RoboDK station: 07252019 KR10 2 Script Print.rdk

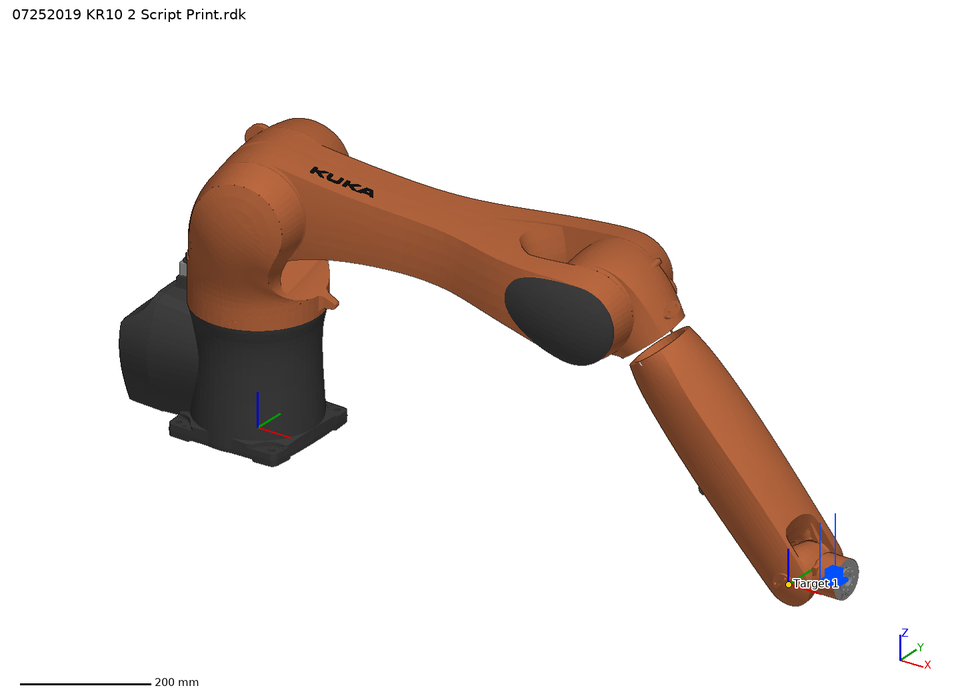
[picture v0: the station drawn from its stored meshes, robots at their saved joint values, targets as dots, program paths as lines]
Station 07252019 KR10 2 Script Print. Poses are relative to the parent item; angles as X-Y-Z fixed-axis rotations.
  - frame KUKA KR 10 R1100 sixx Base at (0, 0, 0) mm
    - robot KUKA KR 10 R1100 sixx: 6 axes, payload 10 kg, reach 1101 mm, repeatability 0.03 mm, weight 54 kg
        modified DH rows (alpha deg, a mm, theta deg, d mm): 0, 0, 0, 400; -90, 25, 0, 0; 0, 560, -90, 0; -90, 35, 0, 515; 90, 0, 0, 0; -90, 0, 180, 80
        joint limits [-170, -190, -120, -185, -120, -350] to [170, 45, 156, 185, 120, 350]; home [0, -90, 90, 0, 0, 0]; saved at [-10.597, 6.174, 47.039, 166.851, 53.94, -172.17]
    - target Target 1 (Cartesian target) at (915.91, 105.12, -52.31) mm, rotated rx -159.1 ry 89.96 rz -159.1 deg; joints [-7.168, 0.501, 63.462, 172.028, 64.143, -176.495] of KUKA KR 10 R1100 sixx
  - frame Frame 2 at (915.91, 105.12, -52.31) mm
  - machining project Print3D settings: C:/Users/Rez/Downloads/XYZ_20mm_Calibration_Cube/files/CFFFP_xyzCalibration_cube.gcode | rotZ(0) | rotX(0)*rotY(0)
  - Python program Extruder (listed below)
  - Python program M_RunCode (listed below)
  - program Print3D (7039 instructions, listed below)
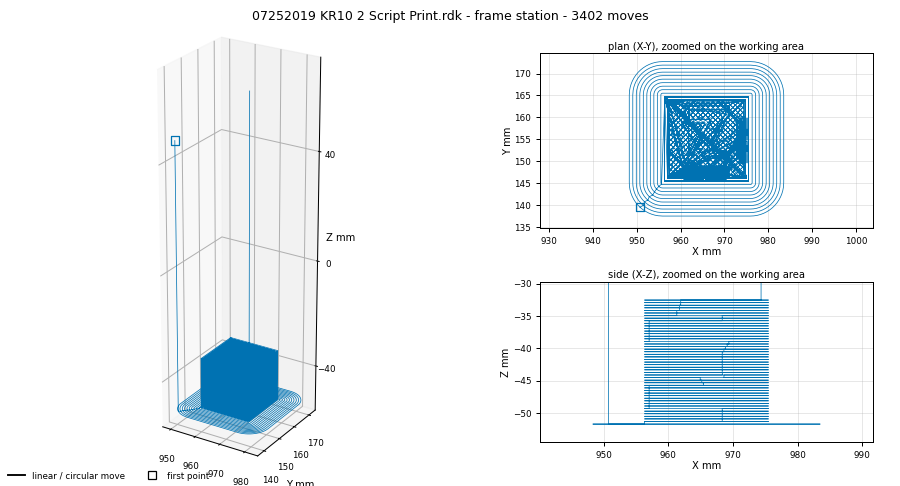
[picture p0: tool path of 07252019 KR10 2 Script Print.rdk in frame station, 3402 of 3402 moves have a stored position in this frame; points joined in program order, loops and branches not executed]

--- Python program Extruder ---
# -*- coding: utf-8 -*-
"""
Created on Fri May 24 11:08:35 2019

@author: Rez
"""

import telnetlib
import sys

tn = telnetlib.Telnet('192.168.1.112', 23)
tn.read_until(b"Smoothie command shell")
str1 = str(sys.argv[1])
str2 = "G1 E" + str1 + "\n"
str3 = str2.encode('utf-8')
tn.write(str3)
tn.read_until(b"ok")
tn.write(b"exit")
tn.close
exit

--- Python program M_RunCode ---
# -*- coding: utf-8 -*-
"""
Created on Fri May 24 11:08:35 2019

@author: Rez
"""

import telnetlib
import sys

tn = telnetlib.Telnet('192.168.1.112', 23)
tn.read_until(b"Smoothie command shell")
str1 = str(sys.argv[1])
str4 = str(sys.argv[2])
str2 = "M" + str1 + " P" +str4 + "\n"
str3 = str2.encode('utf-8')
tn.write(str3)
tn.read_until(b"ok")
tn.write(b"exit")
tn.close
exit

--- program Print3D (robot KUKA KR 10 R1100 sixx) ---
  Accurate (rounding -1 mm)
  Set Ref.: Frame 2
  Set Tool at (0, 0, 0) mm
  Call M_RunCode(104,0)
  Call M_RunCode(105,0)
  Call M_RunCode(109,0)
  Call M_RunCode(82,0)
  Call Extruder(0.000)
  Set speed (3.3 mm/s)
  Call Extruder(0.000)
  Set speed (1000.0 mm/s)
  MoveJ 1 to (34.82, 34.44, 100.6) mm, rotated rx 0 ry 90 rz 0 deg; joints [-9.106, -6.941, 65.166, 169.323, 58.671, -174.401]
  MoveL 2 to (34.82, 34.44, 100.6) mm, rotated rx 0 ry 90 rz 0 deg; joints [-9.106, -6.941, 65.166, 169.323, 58.671, -174.401]
  MoveL 3 to (34.82, 34.44, 0.6) mm, rotated rx 0 ry 90 rz 0 deg; joints [-9.106, 3.069, 55.606, 169.373, 59.113, -174.498]
  MoveL 4 to (34.82, 34.44, 0.6) mm, rotated rx 0 ry 90 rz 0 deg; joints [-9.106, 3.069, 55.606, 169.373, 59.113, -174.498]
  Call Extruder(0.000)
  Call Extruder(0.000)
  Call Extruder(0.000)
  Set speed (30.0 mm/s)
  Call Extruder(0.000)
  MoveL 5 to (34.82, 34.44, 0.6) mm, rotated rx 0 ry 90 rz 0 deg; joints [-9.106, 3.069, 55.606, 169.373, 59.113, -174.498]
  Call M_RunCode(107,0)
  Set speed (60.0 mm/s)
  MoveL 6 to (34.82, 34.44, 0.6) mm, rotated rx 0 ry 90 rz 0 deg; joints [-9.106, 3.069, 55.606, 169.373, 59.113, -174.498]
  Set speed (30.0 mm/s)
  Call Extruder(0.000)
  MoveL 7 to (34.82, 34.44, 0.6) mm, rotated rx 0 ry 90 rz 0 deg; joints [-9.106, 3.069, 55.606, 169.373, 59.113, -174.498]
  Call Extruder(0.156)
  MoveL 8 to (35.42, 33.94, 0.6) mm, rotated rx 0 ry 90 rz 0 deg; joints [-9.068, 3.107, 55.496, 169.409, 59.039, -174.506]
  Call Extruder(0.311)
  MoveL 9 to (36.06, 33.5, 0.6) mm, rotated rx 0 ry 90 rz 0 deg; joints [-9.033, 3.15, 55.372, 169.441, 58.956, -174.509]
  Call Extruder(0.467)
  MoveL 10 to (36.75, 33.13, 0.6) mm, rotated rx 0 ry 90 rz 0 deg; joints [-9.002, 3.197, 55.237, 169.467, 58.867, -174.509]
  Call Extruder(0.622)
  MoveL 11 to (37.47, 32.83, 0.6) mm, rotated rx 0 ry 90 rz 0 deg; joints [-8.976, 3.248, 55.092, 169.487, 58.772, -174.504]
  Call Extruder(0.778)
  MoveL 12 to (38.22, 32.61, 0.6) mm, rotated rx 0 ry 90 rz 0 deg; joints [-8.954, 3.302, 54.938, 169.501, 58.671, -174.496]
  Call Extruder(0.933)
  MoveL 13 to (38.98, 32.47, 0.6) mm, rotated rx 0 ry 90 rz 0 deg; joints [-8.938, 3.358, 54.777, 169.509, 58.566, -174.484]
  Call Extruder(1.137)
  MoveL 14 to (40, 32.4, 0.6) mm, rotated rx 0 ry 90 rz 0 deg; joints [-8.923, 3.435, 54.558, 169.51, 58.425, -174.463]
  Call Extruder(5.128)
  MoveL 15 to (60, 32.4, 0.6) mm, rotated rx 0 ry 90 rz 0 deg; joints [-8.727, 5.076, 49.99, 169.395, 55.528, -173.951]
  Call Extruder(5.284)
  MoveL 16 to (60.78, 32.44, 0.6) mm, rotated rx 0 ry 90 rz 0 deg; joints [-8.722, 5.145, 49.802, 169.386, 55.411, -173.927]
  Call Extruder(5.439)
  MoveL 17 to (61.55, 32.56, 0.6) mm, rotated rx 0 ry 90 rz 0 deg; joints [-8.722, 5.215, 49.612, 169.37, 55.293, -173.9]
  Call Extruder(5.595)
  MoveL 18 to (62.3, 32.76, 0.6) mm, rotated rx 0 ry 90 rz 0 deg; joints [-8.727, 5.285, 49.422, 169.349, 55.175, -173.87]
  Call Extruder(5.750)
  MoveL 19 to (63.03, 33.03, 0.6) mm, rotated rx 0 ry 90 rz 0 deg; joints [-8.737, 5.355, 49.234, 169.321, 55.06, -173.836]
  Call Extruder(5.906)
  MoveL 20 to (63.73, 33.38, 0.6) mm, rotated rx 0 ry 90 rz 0 deg; joints [-8.752, 5.423, 49.051, 169.288, 54.948, -173.8]
  Call Extruder(6.061)
  MoveL 21 to (64.39, 33.8, 0.6) mm, rotated rx 0 ry 90 rz 0 deg; joints [-8.772, 5.488, 48.874, 169.25, 54.841, -173.761]
  Call Extruder(6.217)
  MoveL 22 to (65, 34.28, 0.6) mm, rotated rx 0 ry 90 rz 0 deg; joints [-8.796, 5.551, 48.705, 169.206, 54.739, -173.719]
  Call Extruder(6.372)
  MoveL 23 to (65.56, 34.82, 0.6) mm, rotated rx 0 ry 90 rz 0 deg; joints [-8.824, 5.61, 48.546, 169.159, 54.644, -173.676]
  Call Extruder(6.528)
  MoveL 24 to (66.06, 35.42, 0.6) mm, rotated rx 0 ry 90 rz 0 deg; joints [-8.856, 5.665, 48.398, 169.107, 54.557, -173.632]
  Call Extruder(6.684)
  MoveL 25 to (66.5, 36.06, 0.6) mm, rotated rx 0 ry 90 rz 0 deg; joints [-8.892, 5.714, 48.265, 169.052, 54.478, -173.587]
  Call Extruder(6.839)
  MoveL 26 to (66.87, 36.75, 0.6) mm, rotated rx 0 ry 90 rz 0 deg; joints [-8.931, 5.759, 48.146, 168.994, 54.41, -173.542]
  Call Extruder(6.995)
  MoveL 27 to (67.17, 37.47, 0.6) mm, rotated rx 0 ry 90 rz 0 deg; joints [-8.973, 5.797, 48.044, 168.935, 54.351, -173.498]
  Call Extruder(7.150)
  MoveL 28 to (67.39, 38.22, 0.6) mm, rotated rx 0 ry 90 rz 0 deg; joints [-9.017, 5.829, 47.959, 168.873, 54.304, -173.453]
  Call Extruder(7.306)
  MoveL 29 to (67.53, 38.98, 0.6) mm, rotated rx 0 ry 90 rz 0 deg; joints [-9.063, 5.854, 47.892, 168.811, 54.268, -173.411]
  Call Extruder(7.509)
  MoveL 30 to (67.6, 40, 0.6) mm, rotated rx 0 ry 90 rz 0 deg; joints [-9.125, 5.875, 47.834, 168.73, 54.24, -173.358]
  Call Extruder(11.501)
  MoveL 31 to (67.6, 60, 0.6) mm, rotated rx 0 ry 90 rz 0 deg; joints [-10.357, 6.202, 46.965, 167.138, 53.863, -172.331]
  Call Extruder(11.656)
  MoveL 32 to (67.56, 60.78, 0.6) mm, rotated rx 0 ry 90 rz 0 deg; joints [-10.405, 6.212, 46.939, 167.076, 53.853, -172.292]
  Call Extruder(11.812)
  MoveL 33 to (67.44, 61.55, 0.6) mm, rotated rx 0 ry 90 rz 0 deg; joints [-10.454, 6.214, 46.933, 167.016, 53.856, -172.255]
  Call Extruder(11.967)
  MoveL 34 to (67.24, 62.3, 0.6) mm, rotated rx 0 ry 90 rz 0 deg; joints [-10.502, 6.208, 46.948, 166.958, 53.872, -172.223]
  Call Extruder(12.123)
  MoveL 35 to (66.97, 63.03, 0.6) mm, rotated rx 0 ry 90 rz 0 deg; joints [-10.55, 6.195, 46.983, 166.903, 53.9, -172.194]
  Call Extruder(12.278)
  MoveL 36 to (66.62, 63.73, 0.6) mm, rotated rx 0 ry 90 rz 0 deg; joints [-10.597, 6.174, 47.039, 166.851, 53.94, -172.17]
  Call Extruder(12.434)
  MoveL 37 to (66.21, 64.39, 0.6) mm, rotated rx 0 ry 90 rz 0 deg; joints [-10.642, 6.146, 47.113, 166.803, 53.991, -172.151]
  Call Extruder(12.589)
  MoveL 38 to (65.72, 65, 0.6) mm, rotated rx 0 ry 90 rz 0 deg; joints [-10.685, 6.111, 47.207, 166.76, 54.054, -172.136]
  Call Extruder(12.745)
  MoveL 39 to (65.18, 65.56, 0.6) mm, rotated rx 0 ry 90 rz 0 deg; joints [-10.726, 6.069, 47.317, 166.722, 54.126, -172.127]
  Call Extruder(12.901)
  MoveL 40 to (64.58, 66.06, 0.6) mm, rotated rx 0 ry 90 rz 0 deg; joints [-10.764, 6.022, 47.443, 166.689, 54.209, -172.122]
  Call Extruder(13.056)
  MoveL 41 to (63.94, 66.5, 0.6) mm, rotated rx 0 ry 90 rz 0 deg; joints [-10.798, 5.969, 47.585, 166.662, 54.299, -172.123]
  Call Extruder(13.212)
  MoveL 42 to (63.25, 66.87, 0.6) mm, rotated rx 0 ry 90 rz 0 deg; joints [-10.829, 5.911, 47.739, 166.64, 54.397, -172.128]
  Call Extruder(13.367)
  MoveL 43 to (62.53, 67.17, 0.6) mm, rotated rx 0 ry 90 rz 0 deg; joints [-10.856, 5.849, 47.905, 166.625, 54.502, -172.139]
  Call Extruder(13.523)
  MoveL 44 to (61.78, 67.39, 0.6) mm, rotated rx 0 ry 90 rz 0 deg; joints [-10.878, 5.783, 48.08, 166.615, 54.612, -172.154]
  Call Extruder(13.678)
  MoveL 45 to (61.02, 67.53, 0.6) mm, rotated rx 0 ry 90 rz 0 deg; joints [-10.896, 5.715, 48.263, 166.612, 54.726, -172.174]
  Call Extruder(13.882)
  MoveL 46 to (60, 67.6, 0.6) mm, rotated rx 0 ry 90 rz 0 deg; joints [-10.912, 5.623, 48.511, 166.618, 54.879, -172.207]
  Call Extruder(17.873)
  MoveL 47 to (40, 67.6, 0.6) mm, rotated rx 0 ry 90 rz 0 deg; joints [-11.155, 3.921, 53.184, 166.784, 57.802, -172.867]
  Call Extruder(18.029)
  MoveL 48 to (39.22, 67.56, 0.6) mm, rotated rx 0 ry 90 rz 0 deg; joints [-11.162, 3.859, 53.359, 166.792, 57.913, -172.893]
  Call Extruder(18.184)
  MoveL 49 to (38.45, 67.44, 0.6) mm, rotated rx 0 ry 90 rz 0 deg; joints [-11.164, 3.796, 53.535, 166.805, 58.024, -172.922]
  Call Extruder(18.340)
  MoveL 50 to (37.7, 67.24, 0.6) mm, rotated rx 0 ry 90 rz 0 deg; joints [-11.161, 3.734, 53.71, 166.825, 58.133, -172.955]
  Call Extruder(18.495)
  MoveL 51 to (36.97, 66.97, 0.6) mm, rotated rx 0 ry 90 rz 0 deg; joints [-11.153, 3.673, 53.882, 166.85, 58.24, -172.99]
  Call Extruder(18.651)
  MoveL 52 to (36.27, 66.62, 0.6) mm, rotated rx 0 ry 90 rz 0 deg; joints [-11.14, 3.614, 54.05, 166.881, 58.345, -173.027]
  Call Extruder(18.806)
  MoveL 53 to (35.61, 66.2, 0.6) mm, rotated rx 0 ry 90 rz 0 deg; joints [-11.122, 3.557, 54.212, 166.917, 58.444, -173.066]
  Call Extruder(18.962)
  MoveL 54 to (35, 65.72, 0.6) mm, rotated rx 0 ry 90 rz 0 deg; joints [-11.099, 3.502, 54.366, 166.957, 58.539, -173.106]
  Call Extruder(19.117)
  MoveL 55 to (34.44, 65.18, 0.6) mm, rotated rx 0 ry 90 rz 0 deg; joints [-11.071, 3.452, 54.51, 167.002, 58.627, -173.148]
  Call Extruder(19.273)
  MoveL 56 to (33.94, 64.58, 0.6) mm, rotated rx 0 ry 90 rz 0 deg; joints [-11.04, 3.405, 54.644, 167.051, 58.708, -173.19]
  Call Extruder(19.429)
  MoveL 57 to (33.5, 63.94, 0.6) mm, rotated rx 0 ry 90 rz 0 deg; joints [-11.004, 3.362, 54.766, 167.103, 58.781, -173.232]
  Call Extruder(19.584)
  MoveL 58 to (33.13, 63.25, 0.6) mm, rotated rx 0 ry 90 rz 0 deg; joints [-10.965, 3.324, 54.874, 167.158, 58.845, -173.273]
  Call Extruder(19.740)
  MoveL 59 to (32.83, 62.53, 0.6) mm, rotated rx 0 ry 90 rz 0 deg; joints [-10.923, 3.291, 54.968, 167.215, 58.899, -173.315]
  Call Extruder(19.895)
  MoveL 60 to (32.61, 61.78, 0.6) mm, rotated rx 0 ry 90 rz 0 deg; joints [-10.878, 3.264, 55.047, 167.274, 58.944, -173.355]
  Call Extruder(20.051)
  MoveL 61 to (32.47, 61.02, 0.6) mm, rotated rx 0 ry 90 rz 0 deg; joints [-10.831, 3.242, 55.109, 167.333, 58.978, -173.393]
  Call Extruder(20.254)
  MoveL 62 to (32.4, 60, 0.6) mm, rotated rx 0 ry 90 rz 0 deg; joints [-10.767, 3.222, 55.166, 167.412, 59.007, -173.441]
  Call Extruder(24.246)
  MoveL 63 to (32.4, 40, 0.6) mm, rotated rx 0 ry 90 rz 0 deg; joints [-9.488, 2.957, 55.927, 168.954, 59.357, -174.318]
  Call Extruder(24.401)
  MoveL 64 to (32.44, 39.22, 0.6) mm, rotated rx 0 ry 90 rz 0 deg; joints [-9.438, 2.951, 55.946, 169.013, 59.364, -174.35]
  Call Extruder(24.557)
  MoveL 65 to (32.56, 38.45, 0.6) mm, rotated rx 0 ry 90 rz 0 deg; joints [-9.387, 2.95, 55.948, 169.072, 59.36, -174.38]
  Call Extruder(24.712)
  MoveL 66 to (32.76, 37.7, 0.6) mm, rotated rx 0 ry 90 rz 0 deg; joints [-9.337, 2.956, 55.933, 169.129, 59.345, -174.408]
  Call Extruder(24.868)
  MoveL 67 to (33.03, 36.97, 0.6) mm, rotated rx 0 ry 90 rz 0 deg; joints [-9.287, 2.967, 55.9, 169.185, 59.319, -174.433]
  Call Extruder(25.023)
  MoveL 68 to (33.38, 36.27, 0.6) mm, rotated rx 0 ry 90 rz 0 deg; joints [-9.239, 2.984, 55.85, 169.237, 59.283, -174.454]
  Call Extruder(25.179)
  MoveL 69 to (33.79, 35.61, 0.6) mm, rotated rx 0 ry 90 rz 0 deg; joints [-9.192, 3.007, 55.784, 169.286, 59.236, -174.472]
  Call Extruder(25.334)
  MoveL 70 to (34.28, 35, 0.6) mm, rotated rx 0 ry 90 rz 0 deg; joints [-9.148, 3.035, 55.702, 169.332, 59.179, -174.487]
  Call Extruder(25.490)
  MoveL 71 to (34.82, 34.44, 0.6) mm, rotated rx 0 ry 90 rz 0 deg; joints [-9.106, 3.069, 55.606, 169.373, 59.113, -174.498]
  Set speed (60.0 mm/s)
  MoveL 72 to (35.6, 34.81, 0.6) mm, rotated rx 0 ry 90 rz 0 deg; joints [-9.122, 3.132, 55.425, 169.342, 58.999, -174.463]
  Set speed (30.0 mm/s)
  Call Extruder(25.637)
  MoveL 73 to (36.19, 34.37, 0.6) mm, rotated rx 0 ry 90 rz 0 deg; joints [-9.087, 3.17, 55.315, 169.374, 58.925, -174.469]
  Call Extruder(25.784)
  MoveL 74 to (36.82, 33.99, 0.6) mm, rotated rx 0 ry 90 rz 0 deg; joints [-9.057, 3.213, 55.192, 169.401, 58.843, -174.47]
  Call Extruder(25.931)
  MoveL 75 to (37.49, 33.68, 0.6) mm, rotated rx 0 ry 90 rz 0 deg; joints [-9.03, 3.26, 55.058, 169.422, 58.755, -174.467]
  Call Extruder(26.078)
  MoveL 76 to (38.19, 33.45, 0.6) mm, rotated rx 0 ry 90 rz 0 deg; joints [-9.008, 3.31, 54.915, 169.437, 58.661, -174.46]
  Call Extruder(26.226)
  MoveL 77 to (38.91, 33.29, 0.6) mm, rotated rx 0 ry 90 rz 0 deg; joints [-8.991, 3.363, 54.764, 169.446, 58.563, -174.45]
  Call Extruder(26.443)
  MoveL 78 to (40, 33.2, 0.6) mm, rotated rx 0 ry 90 rz 0 deg; joints [-8.974, 3.445, 54.53, 169.449, 58.413, -174.427]
  Call Extruder(30.435)
  MoveL 79 to (60, 33.2, 0.6) mm, rotated rx 0 ry 90 rz 0 deg; joints [-8.777, 5.087, 49.961, 169.332, 55.515, -173.912]
  Call Extruder(30.582)
  MoveL 80 to (60.74, 33.24, 0.6) mm, rotated rx 0 ry 90 rz 0 deg; joints [-8.772, 5.153, 49.782, 169.323, 55.404, -173.89]
  Call Extruder(30.729)
  MoveL 81 to (61.46, 33.36, 0.6) mm, rotated rx 0 ry 90 rz 0 deg; joints [-8.773, 5.219, 49.602, 169.308, 55.292, -173.864]
  Call Extruder(30.876)
  MoveL 82 to (62.17, 33.56, 0.6) mm, rotated rx 0 ry 90 rz 0 deg; joints [-8.778, 5.285, 49.423, 169.287, 55.182, -173.835]
  Call Extruder(31.023)
  MoveL 83 to (62.86, 33.83, 0.6) mm, rotated rx 0 ry 90 rz 0 deg; joints [-8.789, 5.35, 49.246, 169.26, 55.073, -173.802]
  Call Extruder(31.170)
  MoveL 84 to (63.51, 34.18, 0.6) mm, rotated rx 0 ry 90 rz 0 deg; joints [-8.804, 5.414, 49.074, 169.227, 54.968, -173.767]
  Call Extruder(31.317)
  MoveL 85 to (64.12, 34.59, 0.6) mm, rotated rx 0 ry 90 rz 0 deg; joints [-8.824, 5.475, 48.909, 169.189, 54.869, -173.729]
  Call Extruder(31.464)
  MoveL 86 to (64.68, 35.07, 0.6) mm, rotated rx 0 ry 90 rz 0 deg; joints [-8.848, 5.533, 48.753, 169.147, 54.775, -173.69]
  Call Extruder(31.612)
  MoveL 87 to (65.19, 35.6, 0.6) mm, rotated rx 0 ry 90 rz 0 deg; joints [-8.876, 5.587, 48.608, 169.1, 54.688, -173.649]
  Call Extruder(31.759)
  MoveL 88 to (65.63, 36.19, 0.6) mm, rotated rx 0 ry 90 rz 0 deg; joints [-8.908, 5.636, 48.475, 169.05, 54.61, -173.607]
  Call Extruder(31.906)
  MoveL 89 to (66.01, 36.82, 0.6) mm, rotated rx 0 ry 90 rz 0 deg; joints [-8.944, 5.68, 48.356, 168.996, 54.541, -173.564]
  Call Extruder(32.053)
  MoveL 90 to (66.32, 37.49, 0.6) mm, rotated rx 0 ry 90 rz 0 deg; joints [-8.982, 5.719, 48.253, 168.941, 54.482, -173.522]
  Call Extruder(32.200)
  MoveL 91 to (66.56, 38.19, 0.6) mm, rotated rx 0 ry 90 rz 0 deg; joints [-9.023, 5.751, 48.168, 168.883, 54.433, -173.48]
  Call Extruder(32.347)
  MoveL 92 to (66.71, 38.91, 0.6) mm, rotated rx 0 ry 90 rz 0 deg; joints [-9.067, 5.776, 48.1, 168.825, 54.396, -173.439]
  Call Extruder(32.565)
  MoveL 93 to (66.8, 40, 0.6) mm, rotated rx 0 ry 90 rz 0 deg; joints [-9.133, 5.801, 48.034, 168.738, 54.364, -173.382]
  Call Extruder(36.556)
  MoveL 94 to (66.8, 60, 0.6) mm, rotated rx 0 ry 90 rz 0 deg; joints [-10.366, 6.125, 47.169, 167.147, 53.988, -172.359]
  Call Extruder(36.703)
  MoveL 95 to (66.76, 60.74, 0.6) mm, rotated rx 0 ry 90 rz 0 deg; joints [-10.412, 6.134, 47.145, 167.089, 53.979, -172.322]
  Call Extruder(36.850)
  MoveL 96 to (66.64, 61.46, 0.6) mm, rotated rx 0 ry 90 rz 0 deg; joints [-10.458, 6.136, 47.141, 167.032, 53.983, -172.289]
  Call Extruder(36.998)
  MoveL 97 to (66.44, 62.17, 0.6) mm, rotated rx 0 ry 90 rz 0 deg; joints [-10.503, 6.129, 47.158, 166.978, 54, -172.258]
  Call Extruder(37.145)
  MoveL 98 to (66.17, 62.86, 0.6) mm, rotated rx 0 ry 90 rz 0 deg; joints [-10.549, 6.115, 47.195, 166.926, 54.028, -172.232]
  Call Extruder(37.292)
  MoveL 99 to (65.82, 63.51, 0.6) mm, rotated rx 0 ry 90 rz 0 deg; joints [-10.593, 6.094, 47.252, 166.878, 54.069, -172.211]
  Call Extruder(37.439)
  MoveL 100 to (65.41, 64.12, 0.6) mm, rotated rx 0 ry 90 rz 0 deg; joints [-10.635, 6.065, 47.327, 166.834, 54.12, -172.194]
  Call Extruder(37.586)
  MoveL 101 to (64.93, 64.68, 0.6) mm, rotated rx 0 ry 90 rz 0 deg; joints [-10.675, 6.03, 47.421, 166.795, 54.183, -172.182]
  Call Extruder(37.733)
  MoveL 102 to (64.4, 65.19, 0.6) mm, rotated rx 0 ry 90 rz 0 deg; joints [-10.712, 5.988, 47.532, 166.761, 54.256, -172.175]
  Call Extruder(37.880)
  MoveL 103 to (63.81, 65.63, 0.6) mm, rotated rx 0 ry 90 rz 0 deg; joints [-10.746, 5.941, 47.659, 166.732, 54.337, -172.172]
  Call Extruder(38.028)
  MoveL 104 to (63.18, 66.01, 0.6) mm, rotated rx 0 ry 90 rz 0 deg; joints [-10.777, 5.889, 47.799, 166.709, 54.427, -172.175]
  Call Extruder(38.175)
  MoveL 105 to (62.51, 66.32, 0.6) mm, rotated rx 0 ry 90 rz 0 deg; joints [-10.804, 5.832, 47.951, 166.692, 54.523, -172.183]
  Call Extruder(38.322)
  MoveL 106 to (61.81, 66.56, 0.6) mm, rotated rx 0 ry 90 rz 0 deg; joints [-10.826, 5.771, 48.114, 166.682, 54.625, -172.196]
  Call Extruder(38.469)
  MoveL 107 to (61.09, 66.71, 0.6) mm, rotated rx 0 ry 90 rz 0 deg; joints [-10.845, 5.707, 48.285, 166.677, 54.732, -172.214]
  Call Extruder(38.687)
  MoveL 108 to (60, 66.8, 0.6) mm, rotated rx 0 ry 90 rz 0 deg; joints [-10.863, 5.609, 48.549, 166.682, 54.896, -172.248]
  Call Extruder(42.678)
  MoveL 109 to (40, 66.8, 0.6) mm, rotated rx 0 ry 90 rz 0 deg; joints [-11.105, 3.908, 53.219, 166.846, 57.818, -172.905]
  Call Extruder(42.825)
  MoveL 110 to (39.26, 66.76, 0.6) mm, rotated rx 0 ry 90 rz 0 deg; joints [-11.111, 3.85, 53.384, 166.854, 57.923, -172.929]
  Call Extruder(42.972)
  MoveL 111 to (38.54, 66.64, 0.6) mm, rotated rx 0 ry 90 rz 0 deg; joints [-11.113, 3.791, 53.551, 166.867, 58.027, -172.957]
  Call Extruder(43.119)
  MoveL 112 to (37.83, 66.44, 0.6) mm, rotated rx 0 ry 90 rz 0 deg; joints [-11.109, 3.732, 53.716, 166.886, 58.131, -172.988]
  Call Extruder(43.266)
  MoveL 113 to (37.14, 66.17, 0.6) mm, rotated rx 0 ry 90 rz 0 deg; joints [-11.1, 3.674, 53.878, 166.911, 58.232, -173.021]
  Call Extruder(43.414)
  MoveL 114 to (36.49, 65.82, 0.6) mm, rotated rx 0 ry 90 rz 0 deg; joints [-11.087, 3.619, 54.036, 166.942, 58.329, -173.057]
  Call Extruder(43.561)
  MoveL 115 to (35.88, 65.41, 0.6) mm, rotated rx 0 ry 90 rz 0 deg; joints [-11.068, 3.565, 54.187, 166.977, 58.422, -173.094]
  Call Extruder(43.708)
  MoveL 116 to (35.32, 64.93, 0.6) mm, rotated rx 0 ry 90 rz 0 deg; joints [-11.045, 3.515, 54.33, 167.017, 58.51, -173.133]
  Call Extruder(43.855)
  MoveL 117 to (34.81, 64.4, 0.6) mm, rotated rx 0 ry 90 rz 0 deg; joints [-11.017, 3.468, 54.463, 167.061, 58.59, -173.172]
  Call Extruder(44.002)
  MoveL 118 to (34.37, 63.81, 0.6) mm, rotated rx 0 ry 90 rz 0 deg; joints [-10.985, 3.426, 54.584, 167.109, 58.663, -173.212]
  Call Extruder(44.149)
  MoveL 119 to (33.99, 63.18, 0.6) mm, rotated rx 0 ry 90 rz 0 deg; joints [-10.95, 3.388, 54.693, 167.16, 58.728, -173.252]
  Call Extruder(44.296)
  MoveL 120 to (33.68, 62.51, 0.6) mm, rotated rx 0 ry 90 rz 0 deg; joints [-10.911, 3.354, 54.787, 167.213, 58.783, -173.291]
  Call Extruder(44.443)
  MoveL 121 to (33.44, 61.81, 0.6) mm, rotated rx 0 ry 90 rz 0 deg; joints [-10.87, 3.327, 54.867, 167.268, 58.829, -173.33]
  Call Extruder(44.591)
  MoveL 122 to (33.29, 61.09, 0.6) mm, rotated rx 0 ry 90 rz 0 deg; joints [-10.826, 3.304, 54.93, 167.324, 58.864, -173.367]
  Call Extruder(44.808)
  MoveL 123 to (33.2, 60, 0.6) mm, rotated rx 0 ry 90 rz 0 deg; joints [-10.758, 3.282, 54.994, 167.409, 58.896, -173.418]
  Call Extruder(48.799)
  MoveL 124 to (33.2, 40, 0.6) mm, rotated rx 0 ry 90 rz 0 deg; joints [-9.48, 3.016, 55.757, 168.951, 59.247, -174.298]
  Call Extruder(48.947)
  MoveL 125 to (33.24, 39.26, 0.6) mm, rotated rx 0 ry 90 rz 0 deg; joints [-9.432, 3.01, 55.775, 169.007, 59.253, -174.329]
  Call Extruder(49.094)
  MoveL 126 to (33.36, 38.54, 0.6) mm, rotated rx 0 ry 90 rz 0 deg; joints [-9.384, 3.01, 55.775, 169.063, 59.249, -174.357]
  Call Extruder(49.241)
  MoveL 127 to (33.56, 37.83, 0.6) mm, rotated rx 0 ry 90 rz 0 deg; joints [-9.337, 3.016, 55.758, 169.117, 59.233, -174.383]
  Call Extruder(49.388)
  MoveL 128 to (33.83, 37.14, 0.6) mm, rotated rx 0 ry 90 rz 0 deg; joints [-9.29, 3.028, 55.724, 169.169, 59.207, -174.406]
  Call Extruder(49.535)
  MoveL 129 to (34.18, 36.49, 0.6) mm, rotated rx 0 ry 90 rz 0 deg; joints [-9.244, 3.046, 55.673, 169.217, 59.169, -174.425]
  Call Extruder(49.682)
  MoveL 130 to (34.59, 35.88, 0.6) mm, rotated rx 0 ry 90 rz 0 deg; joints [-9.201, 3.069, 55.606, 169.263, 59.122, -174.442]
  Call Extruder(49.829)
  MoveL 131 to (35.07, 35.32, 0.6) mm, rotated rx 0 ry 90 rz 0 deg; joints [-9.16, 3.098, 55.523, 169.304, 59.065, -174.454]
  Call Extruder(49.977)
  MoveL 132 to (35.6, 34.81, 0.6) mm, rotated rx 0 ry 90 rz 0 deg; joints [-9.122, 3.132, 55.425, 169.342, 58.999, -174.463]
  Set speed (60.0 mm/s)
  MoveL 133 to (35.86, 35.66, 0.6) mm, rotated rx 0 ry 90 rz 0 deg; joints [-9.174, 3.161, 55.342, 169.275, 58.951, -174.421]
  Set speed (30.0 mm/s)
  Call Extruder(50.115)
  MoveL 134 to (36.38, 35.21, 0.6) mm, rotated rx 0 ry 90 rz 0 deg; joints [-9.139, 3.195, 55.244, 169.308, 58.885, -174.427]
  Call Extruder(50.253)
  MoveL 135 to (36.96, 34.83, 0.6) mm, rotated rx 0 ry 90 rz 0 deg; joints [-9.109, 3.233, 55.134, 169.335, 58.811, -174.43]
  Call Extruder(50.391)
  MoveL 136 to (37.58, 34.51, 0.6) mm, rotated rx 0 ry 90 rz 0 deg; joints [-9.082, 3.276, 55.011, 169.357, 58.73, -174.429]
  Call Extruder(50.529)
  MoveL 137 to (38.22, 34.27, 0.6) mm, rotated rx 0 ry 90 rz 0 deg; joints [-9.06, 3.322, 54.88, 169.373, 58.644, -174.424]
  Call Extruder(50.668)
  MoveL 138 to (38.9, 34.1, 0.6) mm, rotated rx 0 ry 90 rz 0 deg; joints [-9.043, 3.371, 54.739, 169.384, 58.553, -174.415]
  Call Extruder(50.806)
  MoveL 139 to (39.58, 34.01, 0.6) mm, rotated rx 0 ry 90 rz 0 deg; joints [-9.03, 3.423, 54.593, 169.388, 58.458, -174.402]
  Call Extruder(50.889)
  MoveL 140 to (40, 34, 0.6) mm, rotated rx 0 ry 90 rz 0 deg; joints [-9.025, 3.454, 54.503, 169.387, 58.4, -174.392]
  Call Extruder(54.880)
  MoveL 141 to (60, 34, 0.6) mm, rotated rx 0 ry 90 rz 0 deg; joints [-8.827, 5.098, 49.931, 169.269, 55.502, -173.874]
  Call Extruder(55.018)
  MoveL 142 to (60.69, 34.04, 0.6) mm, rotated rx 0 ry 90 rz 0 deg; joints [-8.823, 5.16, 49.763, 169.261, 55.398, -173.853]
  Call Extruder(55.157)
  MoveL 143 to (61.37, 34.16, 0.6) mm, rotated rx 0 ry 90 rz 0 deg; joints [-8.823, 5.222, 49.594, 169.246, 55.293, -173.828]
  Call Extruder(55.295)
  MoveL 144 to (62.04, 34.36, 0.6) mm, rotated rx 0 ry 90 rz 0 deg; joints [-8.829, 5.284, 49.426, 169.225, 55.189, -173.8]
  Call Extruder(55.433)
  MoveL 145 to (62.67, 34.63, 0.6) mm, rotated rx 0 ry 90 rz 0 deg; joints [-8.84, 5.345, 49.261, 169.199, 55.088, -173.769]
  Call Extruder(55.571)
  MoveL 146 to (63.28, 34.97, 0.6) mm, rotated rx 0 ry 90 rz 0 deg; joints [-8.856, 5.404, 49.102, 169.167, 54.991, -173.735]
  Call Extruder(55.710)
  MoveL 147 to (63.83, 35.38, 0.6) mm, rotated rx 0 ry 90 rz 0 deg; joints [-8.876, 5.46, 48.949, 169.129, 54.899, -173.699]
  Call Extruder(55.848)
  MoveL 148 to (64.34, 35.86, 0.6) mm, rotated rx 0 ry 90 rz 0 deg; joints [-8.9, 5.513, 48.807, 169.088, 54.814, -173.661]
  Call Extruder(55.986)
  MoveL 149 to (64.79, 36.38, 0.6) mm, rotated rx 0 ry 90 rz 0 deg; joints [-8.929, 5.561, 48.676, 169.042, 54.736, -173.622]
  Call Extruder(56.124)
  MoveL 150 to (65.17, 36.96, 0.6) mm, rotated rx 0 ry 90 rz 0 deg; joints [-8.961, 5.605, 48.559, 168.993, 54.667, -173.582]
  Call Extruder(56.262)
  MoveL 151 to (65.49, 37.58, 0.6) mm, rotated rx 0 ry 90 rz 0 deg; joints [-8.996, 5.643, 48.457, 168.942, 54.608, -173.542]
  Call Extruder(56.400)
  MoveL 152 to (65.73, 38.22, 0.6) mm, rotated rx 0 ry 90 rz 0 deg; joints [-9.034, 5.675, 48.371, 168.888, 54.56, -173.503]
  Call Extruder(56.539)
  MoveL 153 to (65.9, 38.9, 0.6) mm, rotated rx 0 ry 90 rz 0 deg; joints [-9.074, 5.7, 48.303, 168.834, 54.522, -173.464]
  Call Extruder(56.677)
  MoveL 154 to (65.99, 39.58, 0.6) mm, rotated rx 0 ry 90 rz 0 deg; joints [-9.115, 5.719, 48.254, 168.779, 54.497, -173.428]
  Call Extruder(56.760)
  MoveL 155 to (66, 40, 0.6) mm, rotated rx 0 ry 90 rz 0 deg; joints [-9.141, 5.726, 48.234, 168.746, 54.488, -173.406]
  Call Extruder(60.751)
  MoveL 156 to (66, 60, 0.6) mm, rotated rx 0 ry 90 rz 0 deg; joints [-10.375, 6.049, 47.371, 167.157, 54.112, -172.388]
  Call Extruder(60.889)
  MoveL 157 to (65.96, 60.69, 0.6) mm, rotated rx 0 ry 90 rz 0 deg; joints [-10.418, 6.057, 47.349, 167.102, 54.105, -172.353]
  Call Extruder(61.028)
  MoveL 158 to (65.84, 61.37, 0.6) mm, rotated rx 0 ry 90 rz 0 deg; joints [-10.461, 6.058, 47.348, 167.049, 54.109, -172.322]
  Call Extruder(61.166)
  MoveL 159 to (65.64, 62.04, 0.6) mm, rotated rx 0 ry 90 rz 0 deg; joints [-10.504, 6.051, 47.367, 166.998, 54.127, -172.294]
  Call Extruder(61.304)
  MoveL 160 to (65.37, 62.67, 0.6) mm, rotated rx 0 ry 90 rz 0 deg; joints [-10.546, 6.036, 47.406, 166.95, 54.156, -172.271]
  Call Extruder(61.442)
  MoveL 161 to (65.03, 63.28, 0.6) mm, rotated rx 0 ry 90 rz 0 deg; joints [-10.587, 6.014, 47.464, 166.906, 54.197, -172.252]
  Call Extruder(61.581)
  MoveL 162 to (64.62, 63.83, 0.6) mm, rotated rx 0 ry 90 rz 0 deg; joints [-10.626, 5.985, 47.541, 166.867, 54.249, -172.237]
  Call Extruder(61.719)
  MoveL 163 to (64.14, 64.34, 0.6) mm, rotated rx 0 ry 90 rz 0 deg; joints [-10.663, 5.95, 47.636, 166.832, 54.312, -172.228]
  Call Extruder(61.857)
  MoveL 164 to (63.62, 64.79, 0.6) mm, rotated rx 0 ry 90 rz 0 deg; joints [-10.697, 5.908, 47.747, 166.802, 54.384, -172.223]
  Call Extruder(61.995)
  MoveL 165 to (63.04, 65.17, 0.6) mm, rotated rx 0 ry 90 rz 0 deg; joints [-10.727, 5.861, 47.873, 166.778, 54.465, -172.224]
  Call Extruder(62.133)
  MoveL 166 to (62.42, 65.49, 0.6) mm, rotated rx 0 ry 90 rz 0 deg; joints [-10.754, 5.809, 48.011, 166.76, 54.553, -172.23]
  Call Extruder(62.271)
  MoveL 167 to (61.78, 65.73, 0.6) mm, rotated rx 0 ry 90 rz 0 deg; joints [-10.776, 5.753, 48.161, 166.747, 54.647, -172.24]
  Call Extruder(62.410)
  MoveL 168 to (61.1, 65.9, 0.6) mm, rotated rx 0 ry 90 rz 0 deg; joints [-10.794, 5.694, 48.319, 166.742, 54.746, -172.255]
  Call Extruder(62.548)
  MoveL 169 to (60.42, 65.99, 0.6) mm, rotated rx 0 ry 90 rz 0 deg; joints [-10.808, 5.633, 48.484, 166.742, 54.849, -172.275]
  Call Extruder(62.631)
  MoveL 170 to (60, 66, 0.6) mm, rotated rx 0 ry 90 rz 0 deg; joints [-10.814, 5.595, 48.586, 166.745, 54.912, -172.289]
  Call Extruder(66.622)
  MoveL 171 to (40, 66, 0.6) mm, rotated rx 0 ry 90 rz 0 deg; joints [-11.054, 3.896, 53.254, 166.908, 57.834, -172.942]
  Call Extruder(66.760)
  MoveL 172 to (39.31, 65.96, 0.6) mm, rotated rx 0 ry 90 rz 0 deg; joints [-11.06, 3.841, 53.409, 166.916, 57.932, -172.965]
  Call Extruder(66.899)
  MoveL 173 to (38.63, 65.84, 0.6) mm, rotated rx 0 ry 90 rz 0 deg; joints [-11.061, 3.785, 53.566, 166.929, 58.03, -172.992]
  Call Extruder(67.037)
  MoveL 174 to (37.96, 65.64, 0.6) mm, rotated rx 0 ry 90 rz 0 deg; joints [-11.057, 3.73, 53.72, 166.948, 58.127, -173.021]
  Call Extruder(67.175)
  MoveL 175 to (37.33, 65.37, 0.6) mm, rotated rx 0 ry 90 rz 0 deg; joints [-11.048, 3.677, 53.872, 166.972, 58.221, -173.053]
  Call Extruder(67.313)
  MoveL 176 to (36.72, 65.03, 0.6) mm, rotated rx 0 ry 90 rz 0 deg; joints [-11.033, 3.625, 54.019, 167.002, 58.312, -173.087]
  Call Extruder(67.452)
  MoveL 177 to (36.17, 64.62, 0.6) mm, rotated rx 0 ry 90 rz 0 deg; joints [-11.014, 3.576, 54.158, 167.037, 58.398, -173.122]
  Call Extruder(67.590)
  MoveL 178 to (35.66, 64.14, 0.6) mm, rotated rx 0 ry 90 rz 0 deg; joints [-10.991, 3.53, 54.289, 167.076, 58.477, -173.159]
  Call Extruder(67.728)
  MoveL 179 to (35.21, 63.62, 0.6) mm, rotated rx 0 ry 90 rz 0 deg; joints [-10.963, 3.487, 54.409, 167.12, 58.55, -173.196]
  Call Extruder(67.866)
  MoveL 180 to (34.83, 63.04, 0.6) mm, rotated rx 0 ry 90 rz 0 deg; joints [-10.931, 3.449, 54.516, 167.166, 58.614, -173.234]
  Call Extruder(68.004)
  MoveL 181 to (34.51, 62.42, 0.6) mm, rotated rx 0 ry 90 rz 0 deg; joints [-10.896, 3.416, 54.611, 167.215, 58.669, -173.271]
  Call Extruder(68.142)
  MoveL 182 to (34.27, 61.78, 0.6) mm, rotated rx 0 ry 90 rz 0 deg; joints [-10.857, 3.389, 54.69, 167.267, 58.715, -173.307]
  Call Extruder(68.281)
  MoveL 183 to (34.1, 61.1, 0.6) mm, rotated rx 0 ry 90 rz 0 deg; joints [-10.817, 3.366, 54.754, 167.319, 58.751, -173.342]
  Call Extruder(68.419)
  MoveL 184 to (34.01, 60.42, 0.6) mm, rotated rx 0 ry 90 rz 0 deg; joints [-10.774, 3.35, 54.801, 167.373, 58.776, -173.376]
  Call Extruder(68.502)
  MoveL 185 to (34, 60, 0.6) mm, rotated rx 0 ry 90 rz 0 deg; joints [-10.748, 3.342, 54.821, 167.405, 58.786, -173.395]
  Call Extruder(72.493)
  MoveL 186 to (34, 40, 0.6) mm, rotated rx 0 ry 90 rz 0 deg; joints [-9.471, 3.075, 55.587, 168.948, 59.137, -174.278]
  Call Extruder(72.631)
  MoveL 187 to (34.04, 39.31, 0.6) mm, rotated rx 0 ry 90 rz 0 deg; joints [-9.426, 3.07, 55.603, 169.001, 59.143, -174.307]
  Call Extruder(72.770)
  MoveL 188 to (34.16, 38.63, 0.6) mm, rotated rx 0 ry 90 rz 0 deg; joints [-9.381, 3.07, 55.602, 169.053, 59.137, -174.334]
  Call Extruder(72.908)
  MoveL 189 to (34.36, 37.96, 0.6) mm, rotated rx 0 ry 90 rz 0 deg; joints [-9.337, 3.077, 55.583, 169.104, 59.121, -174.358]
  Call Extruder(73.046)
  MoveL 190 to (34.63, 37.33, 0.6) mm, rotated rx 0 ry 90 rz 0 deg; joints [-9.293, 3.089, 55.547, 169.152, 59.094, -174.378]
  Call Extruder(73.184)
  MoveL 191 to (34.97, 36.72, 0.6) mm, rotated rx 0 ry 90 rz 0 deg; joints [-9.251, 3.108, 55.494, 169.197, 59.056, -174.396]
  Call Extruder(73.323)
  MoveL 192 to (35.38, 36.17, 0.6) mm, rotated rx 0 ry 90 rz 0 deg; joints [-9.211, 3.131, 55.426, 169.238, 59.008, -174.41]
  Call Extruder(73.461)
  MoveL 193 to (35.86, 35.66, 0.6) mm, rotated rx 0 ry 90 rz 0 deg; joints [-9.174, 3.161, 55.342, 169.275, 58.951, -174.421]
  Set speed (60.0 mm/s)
  MoveL 194 to (36.64, 36.03, 0.6) mm, rotated rx 0 ry 90 rz 0 deg; joints [-9.189, 3.224, 55.161, 169.244, 58.836, -174.386]
  Set speed (30.0 mm/s)
  Call Extruder(73.589)
  MoveL 195 to (37.16, 35.65, 0.6) mm, rotated rx 0 ry 90 rz 0 deg; joints [-9.159, 3.258, 55.063, 169.272, 58.77, -174.39]
  Call Extruder(73.718)
  MoveL 196 to (37.72, 35.33, 0.6) mm, rotated rx 0 ry 90 rz 0 deg; joints [-9.133, 3.297, 54.952, 169.294, 58.697, -174.39]
  Call Extruder(73.847)
  MoveL 197 to (38.31, 35.08, 0.6) mm, rotated rx 0 ry 90 rz 0 deg; joints [-9.111, 3.339, 54.832, 169.311, 58.618, -174.386]
  Call Extruder(73.975)
  MoveL 198 to (38.93, 34.91, 0.6) mm, rotated rx 0 ry 90 rz 0 deg; joints [-9.094, 3.384, 54.703, 169.321, 58.534, -174.378]
  Call Extruder(74.104)
  MoveL 199 to (39.57, 34.82, 0.6) mm, rotated rx 0 ry 90 rz 0 deg; joints [-9.082, 3.432, 54.567, 169.326, 58.447, -174.367]
  Call Extruder(74.189)
  MoveL 200 to (40, 34.8, 0.6) mm, rotated rx 0 ry 90 rz 0 deg; joints [-9.076, 3.464, 54.475, 169.325, 58.387, -174.357]
  Call Extruder(78.180)
  MoveL 201 to (60, 34.8, 0.6) mm, rotated rx 0 ry 90 rz 0 deg; joints [-8.877, 5.109, 49.901, 169.207, 55.489, -173.835]
  Call Extruder(78.309)
  MoveL 202 to (60.64, 34.84, 0.6) mm, rotated rx 0 ry 90 rz 0 deg; joints [-8.873, 5.166, 49.745, 169.199, 55.392, -173.816]
  Call Extruder(78.438)
  MoveL 203 to (61.28, 34.96, 0.6) mm, rotated rx 0 ry 90 rz 0 deg; joints [-8.874, 5.224, 49.588, 169.184, 55.294, -173.792]
  Call Extruder(78.566)
  MoveL 204 to (61.89, 35.16, 0.6) mm, rotated rx 0 ry 90 rz 0 deg; joints [-8.881, 5.282, 49.431, 169.164, 55.198, -173.765]
  Call Extruder(78.695)
  MoveL 205 to (62.48, 35.43, 0.6) mm, rotated rx 0 ry 90 rz 0 deg; joints [-8.892, 5.338, 49.279, 169.138, 55.105, -173.735]
  Call Extruder(78.824)
  MoveL 206 to (63.02, 35.77, 0.6) mm, rotated rx 0 ry 90 rz 0 deg; joints [-8.908, 5.392, 49.133, 169.106, 55.016, -173.703]
  Call Extruder(78.952)
  MoveL 207 to (63.52, 36.18, 0.6) mm, rotated rx 0 ry 90 rz 0 deg; joints [-8.928, 5.443, 48.995, 169.07, 54.933, -173.669]
  Call Extruder(79.081)
  MoveL 208 to (63.97, 36.64, 0.6) mm, rotated rx 0 ry 90 rz 0 deg; joints [-8.953, 5.49, 48.868, 169.029, 54.857, -173.633]
  Call Extruder(79.210)
  MoveL 209 to (64.35, 37.16, 0.6) mm, rotated rx 0 ry 90 rz 0 deg; joints [-8.981, 5.533, 48.753, 168.985, 54.789, -173.596]
  Call Extruder(79.338)
  MoveL 210 to (64.67, 37.72, 0.6) mm, rotated rx 0 ry 90 rz 0 deg; joints [-9.013, 5.57, 48.653, 168.938, 54.731, -173.559]
  Call Extruder(79.467)
  MoveL 211 to (64.92, 38.31, 0.6) mm, rotated rx 0 ry 90 rz 0 deg; joints [-9.047, 5.601, 48.569, 168.889, 54.683, -173.523]
  Call Extruder(79.596)
  MoveL 212 to (65.09, 38.93, 0.6) mm, rotated rx 0 ry 90 rz 0 deg; joints [-9.084, 5.626, 48.502, 168.838, 54.646, -173.487]
  Call Extruder(79.724)
  MoveL 213 to (65.18, 39.57, 0.6) mm, rotated rx 0 ry 90 rz 0 deg; joints [-9.123, 5.644, 48.454, 168.787, 54.621, -173.452]
  Call Extruder(79.809)
  MoveL 214 to (65.2, 40, 0.6) mm, rotated rx 0 ry 90 rz 0 deg; joints [-9.149, 5.652, 48.432, 168.753, 54.611, -173.431]
  Call Extruder(83.801)
  MoveL 215 to (65.2, 60, 0.6) mm, rotated rx 0 ry 90 rz 0 deg; joints [-10.384, 5.973, 47.573, 167.166, 54.236, -172.416]
  Call Extruder(83.929)
  MoveL 216 to (65.16, 60.64, 0.6) mm, rotated rx 0 ry 90 rz 0 deg; joints [-10.424, 5.98, 47.553, 167.115, 54.23, -172.384]
  Call Extruder(84.058)
  MoveL 217 to (65.04, 61.28, 0.6) mm, rotated rx 0 ry 90 rz 0 deg; joints [-10.464, 5.98, 47.554, 167.066, 54.235, -172.355]
  Call Extruder(84.187)
  MoveL 218 to (64.84, 61.89, 0.6) mm, rotated rx 0 ry 90 rz 0 deg; joints [-10.504, 5.972, 47.575, 167.019, 54.253, -172.33]
  Call Extruder(84.315)
  MoveL 219 to (64.57, 62.48, 0.6) mm, rotated rx 0 ry 90 rz 0 deg; joints [-10.543, 5.957, 47.616, 166.976, 54.284, -172.309]
  Call Extruder(84.444)
  MoveL 220 to (64.23, 63.02, 0.6) mm, rotated rx 0 ry 90 rz 0 deg; joints [-10.581, 5.935, 47.676, 166.936, 54.325, -172.293]
  Call Extruder(84.573)
  MoveL 221 to (63.83, 63.52, 0.6) mm, rotated rx 0 ry 90 rz 0 deg; joints [-10.616, 5.905, 47.754, 166.901, 54.378, -172.282]
  Call Extruder(84.701)
  MoveL 222 to (63.36, 63.97, 0.6) mm, rotated rx 0 ry 90 rz 0 deg; joints [-10.649, 5.87, 47.85, 166.87, 54.44, -172.275]
  Call Extruder(84.830)
  MoveL 223 to (62.84, 64.35, 0.6) mm, rotated rx 0 ry 90 rz 0 deg; joints [-10.679, 5.828, 47.96, 166.845, 54.512, -172.273]
  Call Extruder(84.959)
  MoveL 224 to (62.28, 64.67, 0.6) mm, rotated rx 0 ry 90 rz 0 deg; joints [-10.705, 5.782, 48.085, 166.826, 54.591, -172.277]
  Call Extruder(85.087)
  MoveL 225 to (61.69, 64.92, 0.6) mm, rotated rx 0 ry 90 rz 0 deg; joints [-10.727, 5.731, 48.221, 166.813, 54.677, -172.285]
  Call Extruder(85.216)
  MoveL 226 to (61.06, 65.09, 0.6) mm, rotated rx 0 ry 90 rz 0 deg; joints [-10.745, 5.677, 48.367, 166.806, 54.769, -172.298]
  Call Extruder(85.344)
  MoveL 227 to (60.43, 65.18, 0.6) mm, rotated rx 0 ry 90 rz 0 deg; joints [-10.758, 5.62, 48.52, 166.806, 54.864, -172.316]
  Call Extruder(85.430)
  MoveL 228 to (60, 65.2, 0.6) mm, rotated rx 0 ry 90 rz 0 deg; joints [-10.764, 5.581, 48.624, 166.809, 54.928, -172.33]
  Call Extruder(89.421)
  MoveL 229 to (40, 65.2, 0.6) mm, rotated rx 0 ry 90 rz 0 deg; joints [-11.004, 3.884, 53.289, 166.971, 57.849, -172.98]
  Call Extruder(89.550)
  MoveL 230 to (39.36, 65.16, 0.6) mm, rotated rx 0 ry 90 rz 0 deg; joints [-11.009, 3.832, 53.433, 166.978, 57.941, -173.001]
  Call Extruder(89.678)
  MoveL 231 to (38.72, 65.04, 0.6) mm, rotated rx 0 ry 90 rz 0 deg; joints [-11.01, 3.781, 53.579, 166.99, 58.032, -173.026]
  Call Extruder(89.807)
  MoveL 232 to (38.11, 64.84, 0.6) mm, rotated rx 0 ry 90 rz 0 deg; joints [-11.005, 3.73, 53.723, 167.009, 58.122, -173.054]
  Call Extruder(89.936)
  MoveL 233 to (37.52, 64.57, 0.6) mm, rotated rx 0 ry 90 rz 0 deg; joints [-10.995, 3.68, 53.863, 167.033, 58.209, -173.084]
  Call Extruder(90.064)
  MoveL 234 to (36.98, 64.23, 0.6) mm, rotated rx 0 ry 90 rz 0 deg; joints [-10.98, 3.632, 53.997, 167.063, 58.292, -173.116]
  Call Extruder(90.193)
  MoveL 235 to (36.48, 63.83, 0.6) mm, rotated rx 0 ry 90 rz 0 deg; joints [-10.96, 3.588, 54.124, 167.097, 58.37, -173.149]
  Call Extruder(90.321)
  MoveL 236 to (36.03, 63.36, 0.6) mm, rotated rx 0 ry 90 rz 0 deg; joints [-10.936, 3.546, 54.241, 167.135, 58.441, -173.184]
  Call Extruder(90.450)
  MoveL 237 to (35.65, 62.84, 0.6) mm, rotated rx 0 ry 90 rz 0 deg; joints [-10.908, 3.509, 54.347, 167.177, 58.504, -173.219]
  Call Extruder(90.579)
  MoveL 238 to (35.33, 62.28, 0.6) mm, rotated rx 0 ry 90 rz 0 deg; joints [-10.877, 3.476, 54.44, 167.222, 58.559, -173.254]
  Call Extruder(90.708)
  MoveL 239 to (35.08, 61.69, 0.6) mm, rotated rx 0 ry 90 rz 0 deg; joints [-10.842, 3.449, 54.518, 167.27, 58.605, -173.288]
  Call Extruder(90.836)
  MoveL 240 to (34.91, 61.06, 0.6) mm, rotated rx 0 ry 90 rz 0 deg; joints [-10.804, 3.427, 54.581, 167.319, 58.64, -173.321]
  Call Extruder(90.965)
  MoveL 241 to (34.82, 60.43, 0.6) mm, rotated rx 0 ry 90 rz 0 deg; joints [-10.765, 3.411, 54.627, 167.368, 58.665, -173.352]
  Call Extruder(91.050)
  MoveL 242 to (34.8, 60, 0.6) mm, rotated rx 0 ry 90 rz 0 deg; joints [-10.738, 3.403, 54.648, 167.402, 58.675, -173.372]
  Call Extruder(95.041)
  MoveL 243 to (34.8, 40, 0.6) mm, rotated rx 0 ry 90 rz 0 deg; joints [-9.463, 3.135, 55.416, 168.945, 59.026, -174.258]
  Call Extruder(95.170)
  MoveL 244 to (34.84, 39.36, 0.6) mm, rotated rx 0 ry 90 rz 0 deg; joints [-9.421, 3.13, 55.43, 168.995, 59.031, -174.285]
  Call Extruder(95.299)
  MoveL 245 to (34.96, 38.72, 0.6) mm, rotated rx 0 ry 90 rz 0 deg; joints [-9.379, 3.131, 55.427, 169.043, 59.025, -174.31]
  Call Extruder(95.427)
  MoveL 246 to (35.16, 38.11, 0.6) mm, rotated rx 0 ry 90 rz 0 deg; joints [-9.338, 3.138, 55.407, 169.089, 59.008, -174.332]
  Call Extruder(95.556)
  MoveL 247 to (35.43, 37.52, 0.6) mm, rotated rx 0 ry 90 rz 0 deg; joints [-9.297, 3.151, 55.369, 169.134, 58.98, -174.35]
  Call Extruder(95.685)
  MoveL 248 to (35.77, 36.98, 0.6) mm, rotated rx 0 ry 90 rz 0 deg; joints [-9.259, 3.17, 55.315, 169.174, 58.942, -174.366]
  Call Extruder(95.813)
  MoveL 249 to (36.17, 36.48, 0.6) mm, rotated rx 0 ry 90 rz 0 deg; joints [-9.223, 3.194, 55.245, 169.211, 58.893, -174.378]
  Call Extruder(95.942)
  MoveL 250 to (36.64, 36.03, 0.6) mm, rotated rx 0 ry 90 rz 0 deg; joints [-9.189, 3.224, 55.161, 169.244, 58.836, -174.386]
  Set speed (60.0 mm/s)
  MoveL 251 to (36.96, 36.82, 0.6) mm, rotated rx 0 ry 90 rz 0 deg; joints [-9.236, 3.258, 55.063, 169.182, 58.778, -174.343]
  Set speed (30.0 mm/s)
  Call Extruder(96.060)
  MoveL 252 to (37.42, 36.44, 0.6) mm, rotated rx 0 ry 90 rz 0 deg; joints [-9.207, 3.288, 54.978, 169.21, 58.721, -174.349]
  Call Extruder(96.178)
  MoveL 253 to (37.92, 36.12, 0.6) mm, rotated rx 0 ry 90 rz 0 deg; joints [-9.182, 3.322, 54.88, 169.232, 58.656, -174.35]
  Call Extruder(96.297)
  MoveL 254 to (38.46, 35.88, 0.6) mm, rotated rx 0 ry 90 rz 0 deg; joints [-9.161, 3.36, 54.772, 169.249, 58.585, -174.348]
  Call Extruder(96.415)
  MoveL 255 to (39.03, 35.71, 0.6) mm, rotated rx 0 ry 90 rz 0 deg; joints [-9.144, 3.401, 54.654, 169.259, 58.508, -174.341]
  Call Extruder(96.533)
  MoveL 256 to (39.62, 35.62, 0.6) mm, rotated rx 0 ry 90 rz 0 deg; joints [-9.132, 3.445, 54.53, 169.264, 58.428, -174.331]
  Call Extruder(96.610)
  MoveL 257 to (40, 35.6, 0.6) mm, rotated rx 0 ry 90 rz 0 deg; joints [-9.127, 3.474, 54.447, 169.264, 58.374, -174.322]
  Call Extruder(100.601)
  MoveL 258 to (60, 35.6, 0.6) mm, rotated rx 0 ry 90 rz 0 deg; joints [-8.927, 5.12, 49.871, 169.144, 55.476, -173.797]
  Call Extruder(100.720)
  MoveL 259 to (60.59, 35.64, 0.6) mm, rotated rx 0 ry 90 rz 0 deg; joints [-8.923, 5.173, 49.727, 169.136, 55.386, -173.778]
  Call Extruder(100.838)
  MoveL 260 to (61.17, 35.76, 0.6) mm, rotated rx 0 ry 90 rz 0 deg; joints [-8.925, 5.226, 49.583, 169.122, 55.296, -173.756]
  Call Extruder(100.956)
  MoveL 261 to (61.73, 35.96, 0.6) mm, rotated rx 0 ry 90 rz 0 deg; joints [-8.932, 5.279, 49.44, 169.102, 55.209, -173.731]
  Call Extruder(101.075)
  MoveL 262 to (62.26, 36.23, 0.6) mm, rotated rx 0 ry 90 rz 0 deg; joints [-8.944, 5.33, 49.301, 169.077, 55.124, -173.703]
  Call Extruder(101.193)
  MoveL 263 to (62.75, 36.56, 0.6) mm, rotated rx 0 ry 90 rz 0 deg; joints [-8.96, 5.379, 49.17, 169.046, 55.044, -173.672]
  Call Extruder(101.311)
  MoveL 264 to (63.18, 36.96, 0.6) mm, rotated rx 0 ry 90 rz 0 deg; joints [-8.98, 5.424, 49.048, 169.011, 54.971, -173.64]
  Call Extruder(101.430)
  MoveL 265 to (63.56, 37.42, 0.6) mm, rotated rx 0 ry 90 rz 0 deg; joints [-9.005, 5.465, 48.937, 168.972, 54.906, -173.607]
  Call Extruder(101.548)
  MoveL 266 to (63.88, 37.92, 0.6) mm, rotated rx 0 ry 90 rz 0 deg; joints [-9.033, 5.501, 48.84, 168.929, 54.849, -173.573]
  Call Extruder(101.666)
  MoveL 267 to (64.12, 38.46, 0.6) mm, rotated rx 0 ry 90 rz 0 deg; joints [-9.064, 5.531, 48.759, 168.884, 54.802, -173.539]
  Call Extruder(101.785)
  MoveL 268 to (64.29, 39.03, 0.6) mm, rotated rx 0 ry 90 rz 0 deg; joints [-9.098, 5.554, 48.695, 168.838, 54.767, -173.506]
  Call Extruder(101.903)
  MoveL 269 to (64.38, 39.62, 0.6) mm, rotated rx 0 ry 90 rz 0 deg; joints [-9.133, 5.571, 48.649, 168.791, 54.743, -173.474]
  Call Extruder(101.979)
  MoveL 270 to (64.4, 40, 0.6) mm, rotated rx 0 ry 90 rz 0 deg; joints [-9.157, 5.579, 48.63, 168.761, 54.733, -173.455]
  Call Extruder(105.971)
  MoveL 271 to (64.4, 60, 0.6) mm, rotated rx 0 ry 90 rz 0 deg; joints [-10.393, 5.898, 47.774, 167.175, 54.36, -172.444]
  Call Extruder(106.089)
  MoveL 272 to (64.36, 60.59, 0.6) mm, rotated rx 0 ry 90 rz 0 deg; joints [-10.43, 5.904, 47.757, 167.128, 54.354, -172.415]
  Call Extruder(106.207)
  MoveL 273 to (64.24, 61.17, 0.6) mm, rotated rx 0 ry 90 rz 0 deg; joints [-10.467, 5.903, 47.76, 167.083, 54.361, -172.389]
  Call Extruder(106.326)
  MoveL 274 to (64.04, 61.73, 0.6) mm, rotated rx 0 ry 90 rz 0 deg; joints [-10.504, 5.895, 47.783, 167.041, 54.38, -172.367]
  Call Extruder(106.444)
  MoveL 275 to (63.78, 62.26, 0.6) mm, rotated rx 0 ry 90 rz 0 deg; joints [-10.539, 5.878, 47.826, 167.002, 54.411, -172.349]
  Call Extruder(106.562)
  MoveL 276 to (63.44, 62.75, 0.6) mm, rotated rx 0 ry 90 rz 0 deg; joints [-10.573, 5.855, 47.888, 166.967, 54.453, -172.335]
  Call Extruder(106.681)
  MoveL 277 to (63.04, 63.18, 0.6) mm, rotated rx 0 ry 90 rz 0 deg; joints [-10.605, 5.826, 47.967, 166.936, 54.506, -172.327]
  Call Extruder(106.799)
  MoveL 278 to (62.58, 63.56, 0.6) mm, rotated rx 0 ry 90 rz 0 deg; joints [-10.633, 5.79, 48.063, 166.911, 54.568, -172.323]
  Call Extruder(106.917)
  MoveL 279 to (62.08, 63.88, 0.6) mm, rotated rx 0 ry 90 rz 0 deg; joints [-10.658, 5.749, 48.173, 166.892, 54.639, -172.325]
  Call Extruder(107.036)
  MoveL 280 to (61.54, 64.12, 0.6) mm, rotated rx 0 ry 90 rz 0 deg; joints [-10.68, 5.703, 48.295, 166.878, 54.716, -172.331]
  Call Extruder(107.154)
  MoveL 281 to (60.97, 64.29, 0.6) mm, rotated rx 0 ry 90 rz 0 deg; joints [-10.697, 5.654, 48.428, 166.871, 54.8, -172.342]
  Call Extruder(107.272)
  MoveL 282 to (60.38, 64.38, 0.6) mm, rotated rx 0 ry 90 rz 0 deg; joints [-10.709, 5.602, 48.568, 166.87, 54.887, -172.358]
  Call Extruder(107.349)
  MoveL 283 to (60, 64.4, 0.6) mm, rotated rx 0 ry 90 rz 0 deg; joints [-10.715, 5.567, 48.661, 166.872, 54.945, -172.371]
  Call Extruder(111.340)
  MoveL 284 to (40, 64.4, 0.6) mm, rotated rx 0 ry 90 rz 0 deg; joints [-10.954, 3.871, 53.323, 167.033, 57.865, -173.017]
  Call Extruder(111.459)
  MoveL 285 to (39.41, 64.36, 0.6) mm, rotated rx 0 ry 90 rz 0 deg; joints [-10.958, 3.824, 53.456, 167.039, 57.949, -173.037]
  Call Extruder(111.577)
  MoveL 286 to (38.83, 64.24, 0.6) mm, rotated rx 0 ry 90 rz 0 deg; joints [-10.958, 3.777, 53.59, 167.052, 58.033, -173.06]
  Call Extruder(111.695)
  MoveL 287 to (38.27, 64.05, 0.6) mm, rotated rx 0 ry 90 rz 0 deg; joints [-10.952, 3.73, 53.722, 167.07, 58.115, -173.086]
  Call Extruder(111.813)
  MoveL 288 to (37.74, 63.78, 0.6) mm, rotated rx 0 ry 90 rz 0 deg; joints [-10.942, 3.685, 53.849, 167.094, 58.194, -173.114]
  Call Extruder(111.932)
  MoveL 289 to (37.25, 63.44, 0.6) mm, rotated rx 0 ry 90 rz 0 deg; joints [-10.926, 3.642, 53.971, 167.123, 58.269, -173.144]
  Call Extruder(112.050)
  MoveL 290 to (36.82, 63.04, 0.6) mm, rotated rx 0 ry 90 rz 0 deg; joints [-10.906, 3.602, 54.083, 167.156, 58.338, -173.175]
  Call Extruder(112.168)
  MoveL 291 to (36.44, 62.58, 0.6) mm, rotated rx 0 ry 90 rz 0 deg; joints [-10.882, 3.566, 54.186, 167.194, 58.399, -173.208]
  Call Extruder(112.287)
  MoveL 292 to (36.12, 62.08, 0.6) mm, rotated rx 0 ry 90 rz 0 deg; joints [-10.854, 3.534, 54.275, 167.234, 58.452, -173.24]
  Call Extruder(112.405)
  MoveL 293 to (35.88, 61.54, 0.6) mm, rotated rx 0 ry 90 rz 0 deg; joints [-10.823, 3.508, 54.351, 167.277, 58.497, -173.271]
  Call Extruder(112.524)
  MoveL 294 to (35.71, 60.97, 0.6) mm, rotated rx 0 ry 90 rz 0 deg; joints [-10.789, 3.486, 54.411, 167.322, 58.531, -173.302]
  Call Extruder(112.642)
  MoveL 295 to (35.62, 60.38, 0.6) mm, rotated rx 0 ry 90 rz 0 deg; joints [-10.753, 3.471, 54.455, 167.368, 58.555, -173.331]
  Call Extruder(112.718)
  MoveL 296 to (35.6, 60, 0.6) mm, rotated rx 0 ry 90 rz 0 deg; joints [-10.729, 3.464, 54.475, 167.398, 58.564, -173.349]
  Call Extruder(116.710)
  MoveL 297 to (35.6, 40, 0.6) mm, rotated rx 0 ry 90 rz 0 deg; joints [-9.454, 3.195, 55.244, 168.942, 58.916, -174.238]
  Call Extruder(116.828)
  MoveL 298 to (35.64, 39.41, 0.6) mm, rotated rx 0 ry 90 rz 0 deg; joints [-9.416, 3.19, 55.257, 168.988, 58.92, -174.263]
  Call Extruder(116.946)
  MoveL 299 to (35.76, 38.83, 0.6) mm, rotated rx 0 ry 90 rz 0 deg; joints [-9.377, 3.192, 55.252, 169.032, 58.913, -174.286]
  Call Extruder(117.065)
  MoveL 300 to (35.95, 38.27, 0.6) mm, rotated rx 0 ry 90 rz 0 deg; joints [-9.34, 3.2, 55.229, 169.074, 58.895, -174.305]
  Call Extruder(117.183)
  MoveL 301 to (36.22, 37.74, 0.6) mm, rotated rx 0 ry 90 rz 0 deg; joints [-9.303, 3.214, 55.19, 169.114, 58.866, -174.321]
  Call Extruder(117.301)
  MoveL 302 to (36.56, 37.25, 0.6) mm, rotated rx 0 ry 90 rz 0 deg; joints [-9.268, 3.233, 55.134, 169.15, 58.827, -174.334]
  Call Extruder(117.420)
  MoveL 303 to (36.96, 36.82, 0.6) mm, rotated rx 0 ry 90 rz 0 deg; joints [-9.236, 3.258, 55.063, 169.182, 58.778, -174.343]
  Set speed (60.0 mm/s)
  MoveL 304 to (37.75, 37.19, 0.6) mm, rotated rx 0 ry 90 rz 0 deg; joints [-9.252, 3.322, 54.881, 169.15, 58.663, -174.308]
  Set speed (30.0 mm/s)
  Call Extruder(117.527)
  MoveL 305 to (38.19, 36.89, 0.6) mm, rotated rx 0 ry 90 rz 0 deg; joints [-9.228, 3.352, 54.796, 169.172, 58.607, -174.31]
  Call Extruder(117.634)
  MoveL 306 to (38.67, 36.65, 0.6) mm, rotated rx 0 ry 90 rz 0 deg; joints [-9.208, 3.385, 54.699, 169.188, 58.543, -174.308]
  Call Extruder(117.741)
  MoveL 307 to (39.18, 36.49, 0.6) mm, rotated rx 0 ry 90 rz 0 deg; joints [-9.193, 3.422, 54.594, 169.198, 58.474, -174.303]
  Call Extruder(117.848)
  MoveL 308 to (39.71, 36.41, 0.6) mm, rotated rx 0 ry 90 rz 0 deg; joints [-9.182, 3.462, 54.481, 169.202, 58.401, -174.293]
  Call Extruder(117.905)
  MoveL 309 to (40, 36.4, 0.6) mm, rotated rx 0 ry 90 rz 0 deg; joints [-9.178, 3.484, 54.419, 169.202, 58.361, -174.287]
  Call Extruder(121.896)
  MoveL 310 to (60, 36.4, 0.6) mm, rotated rx 0 ry 90 rz 0 deg; joints [-8.977, 5.131, 49.841, 169.081, 55.462, -173.758]
  Call Extruder(122.003)
  MoveL 311 to (60.53, 36.44, 0.6) mm, rotated rx 0 ry 90 rz 0 deg; joints [-8.974, 5.179, 49.71, 169.074, 55.381, -173.741]
  Call Extruder(122.110)
  MoveL 312 to (61.06, 36.56, 0.6) mm, rotated rx 0 ry 90 rz 0 deg; joints [-8.976, 5.227, 49.58, 169.06, 55.3, -173.721]
  Call Extruder(122.217)
  MoveL 313 to (61.56, 36.75, 0.6) mm, rotated rx 0 ry 90 rz 0 deg; joints [-8.983, 5.274, 49.452, 169.041, 55.222, -173.697]
  Call Extruder(122.324)
  MoveL 314 to (62.02, 37.02, 0.6) mm, rotated rx 0 ry 90 rz 0 deg; joints [-8.995, 5.32, 49.328, 169.016, 55.147, -173.671]
  Call Extruder(122.431)
  MoveL 315 to (62.44, 37.35, 0.6) mm, rotated rx 0 ry 90 rz 0 deg; joints [-9.012, 5.362, 49.213, 168.986, 55.077, -173.642]
  Call Extruder(122.538)
  MoveL 316 to (62.81, 37.75, 0.6) mm, rotated rx 0 ry 90 rz 0 deg; joints [-9.033, 5.401, 49.109, 168.952, 55.015, -173.613]
  Call Extruder(122.645)
  MoveL 317 to (63.11, 38.19, 0.6) mm, rotated rx 0 ry 90 rz 0 deg; joints [-9.057, 5.435, 49.018, 168.915, 54.961, -173.582]
  Call Extruder(122.752)
  MoveL 318 to (63.35, 38.67, 0.6) mm, rotated rx 0 ry 90 rz 0 deg; joints [-9.085, 5.463, 48.941, 168.875, 54.917, -173.551]
  Call Extruder(122.859)
  MoveL 319 to (63.51, 39.18, 0.6) mm, rotated rx 0 ry 90 rz 0 deg; joints [-9.115, 5.485, 48.882, 168.833, 54.884, -173.522]
  Call Extruder(122.966)
  MoveL 320 to (63.59, 39.71, 0.6) mm, rotated rx 0 ry 90 rz 0 deg; joints [-9.147, 5.5, 48.841, 168.791, 54.862, -173.493]
  Call Extruder(123.024)
  MoveL 321 to (63.6, 40, 0.6) mm, rotated rx 0 ry 90 rz 0 deg; joints [-9.165, 5.506, 48.827, 168.768, 54.856, -173.479]
  Call Extruder(127.015)
  MoveL 322 to (63.6, 60, 0.6) mm, rotated rx 0 ry 90 rz 0 deg; joints [-10.402, 5.823, 47.974, 167.184, 54.483, -172.471]
  Call Extruder(127.122)
  MoveL 323 to (63.56, 60.53, 0.6) mm, rotated rx 0 ry 90 rz 0 deg; joints [-10.435, 5.829, 47.959, 167.142, 54.479, -172.445]
  Call Extruder(127.229)
  MoveL 324 to (63.44, 61.06, 0.6) mm, rotated rx 0 ry 90 rz 0 deg; joints [-10.469, 5.826, 47.965, 167.101, 54.487, -172.422]
  Call Extruder(127.336)
  MoveL 325 to (63.25, 61.56, 0.6) mm, rotated rx 0 ry 90 rz 0 deg; joints [-10.502, 5.817, 47.99, 167.064, 54.506, -172.404]
  Call Extruder(127.443)
  MoveL 326 to (62.98, 62.02, 0.6) mm, rotated rx 0 ry 90 rz 0 deg; joints [-10.534, 5.8, 48.036, 167.03, 54.538, -172.389]
  Call Extruder(127.550)
  MoveL 327 to (62.65, 62.44, 0.6) mm, rotated rx 0 ry 90 rz 0 deg; joints [-10.563, 5.776, 48.099, 167, 54.581, -172.379]
  Call Extruder(127.657)
  MoveL 328 to (62.25, 62.81, 0.6) mm, rotated rx 0 ry 90 rz 0 deg; joints [-10.59, 5.746, 48.179, 166.975, 54.634, -172.374]
  Call Extruder(127.764)
  MoveL 329 to (61.81, 63.11, 0.6) mm, rotated rx 0 ry 90 rz 0 deg; joints [-10.614, 5.711, 48.275, 166.956, 54.695, -172.374]
  Call Extruder(127.871)
  MoveL 330 to (61.33, 63.35, 0.6) mm, rotated rx 0 ry 90 rz 0 deg; joints [-10.634, 5.67, 48.383, 166.942, 54.764, -172.378]
  Call Extruder(127.978)
  MoveL 331 to (60.82, 63.51, 0.6) mm, rotated rx 0 ry 90 rz 0 deg; joints [-10.65, 5.626, 48.502, 166.935, 54.839, -172.388]
  Call Extruder(128.085)
  MoveL 332 to (60.29, 63.59, 0.6) mm, rotated rx 0 ry 90 rz 0 deg; joints [-10.661, 5.579, 48.628, 166.934, 54.917, -172.402]
  Call Extruder(128.142)
  MoveL 333 to (60, 63.6, 0.6) mm, rotated rx 0 ry 90 rz 0 deg; joints [-10.665, 5.553, 48.698, 166.936, 54.961, -172.411]
  Call Extruder(132.134)
  MoveL 334 to (40, 63.6, 0.6) mm, rotated rx 0 ry 90 rz 0 deg; joints [-10.903, 3.859, 53.358, 167.095, 57.88, -173.054]
  Call Extruder(132.241)
  MoveL 335 to (39.47, 63.56, 0.6) mm, rotated rx 0 ry 90 rz 0 deg; joints [-10.907, 3.816, 53.478, 167.101, 57.956, -173.072]
  Call Extruder(132.348)
  MoveL 336 to (38.94, 63.44, 0.6) mm, rotated rx 0 ry 90 rz 0 deg; joints [-10.906, 3.774, 53.599, 167.114, 58.032, -173.094]
  Call Extruder(132.455)
  MoveL 337 to (38.44, 63.25, 0.6) mm, rotated rx 0 ry 90 rz 0 deg; joints [-10.9, 3.732, 53.717, 167.131, 58.106, -173.118]
  Call Extruder(132.562)
  MoveL 338 to (37.98, 62.98, 0.6) mm, rotated rx 0 ry 90 rz 0 deg; joints [-10.888, 3.691, 53.831, 167.155, 58.176, -173.144]
  Call Extruder(132.669)
  MoveL 339 to (37.56, 62.64, 0.6) mm, rotated rx 0 ry 90 rz 0 deg; joints [-10.872, 3.654, 53.937, 167.183, 58.241, -173.172]
  Call Extruder(132.776)
  MoveL 340 to (37.19, 62.25, 0.6) mm, rotated rx 0 ry 90 rz 0 deg; joints [-10.852, 3.619, 54.034, 167.215, 58.3, -173.2]
  Call Extruder(132.883)
  MoveL 341 to (36.89, 61.81, 0.6) mm, rotated rx 0 ry 90 rz 0 deg; joints [-10.828, 3.59, 54.119, 167.251, 58.351, -173.229]
  Call Extruder(132.990)
  MoveL 342 to (36.65, 61.33, 0.6) mm, rotated rx 0 ry 90 rz 0 deg; joints [-10.8, 3.564, 54.19, 167.29, 58.393, -173.258]
  Call Extruder(133.097)
  MoveL 343 to (36.49, 60.82, 0.6) mm, rotated rx 0 ry 90 rz 0 deg; joints [-10.77, 3.544, 54.246, 167.33, 58.425, -173.286]
  Call Extruder(133.204)
  MoveL 344 to (36.41, 60.29, 0.6) mm, rotated rx 0 ry 90 rz 0 deg; joints [-10.737, 3.53, 54.287, 167.372, 58.446, -173.313]
  Call Extruder(133.261)
  MoveL 345 to (36.4, 60, 0.6) mm, rotated rx 0 ry 90 rz 0 deg; joints [-10.719, 3.525, 54.301, 167.394, 58.453, -173.326]
  Call Extruder(137.252)
  MoveL 346 to (36.4, 40, 0.6) mm, rotated rx 0 ry 90 rz 0 deg; joints [-9.446, 3.255, 55.072, 168.939, 58.805, -174.218]
  Call Extruder(137.359)
  MoveL 347 to (36.44, 39.46, 0.6) mm, rotated rx 0 ry 90 rz 0 deg; joints [-9.411, 3.251, 55.083, 168.98, 58.808, -174.241]
  Call Extruder(137.466)
  MoveL 348 to (36.56, 38.94, 0.6) mm, rotated rx 0 ry 90 rz 0 deg; joints [-9.376, 3.254, 55.075, 169.02, 58.8, -174.261]
  Call Extruder(137.573)
  MoveL 349 to (36.75, 38.44, 0.6) mm, rotated rx 0 ry 90 rz 0 deg; joints [-9.342, 3.262, 55.051, 169.058, 58.781, -174.278]
  Call Extruder(137.680)
  MoveL 350 to (37.02, 37.98, 0.6) mm, rotated rx 0 ry 90 rz 0 deg; joints [-9.31, 3.277, 55.01, 169.092, 58.752, -174.291]
  Call Extruder(137.787)
  MoveL 351 to (37.35, 37.56, 0.6) mm, rotated rx 0 ry 90 rz 0 deg; joints [-9.279, 3.297, 54.953, 169.124, 58.712, -174.301]
  Call Extruder(137.894)
  MoveL 352 to (37.75, 37.19, 0.6) mm, rotated rx 0 ry 90 rz 0 deg; joints [-9.252, 3.322, 54.881, 169.15, 58.663, -174.308]
  Set speed (60.0 mm/s)
  MoveL 353 to (38.14, 37.91, 0.6) mm, rotated rx 0 ry 90 rz 0 deg; joints [-9.293, 3.361, 54.77, 169.094, 58.597, -174.267]
  Set speed (30.0 mm/s)
  Call Extruder(137.989)
  MoveL 354 to (38.52, 37.62, 0.6) mm, rotated rx 0 ry 90 rz 0 deg; joints [-9.271, 3.386, 54.698, 169.114, 58.549, -174.27]
  Call Extruder(138.083)
  MoveL 355 to (38.94, 37.41, 0.6) mm, rotated rx 0 ry 90 rz 0 deg; joints [-9.253, 3.415, 54.614, 169.129, 58.493, -174.269]
  Call Extruder(138.178)
  MoveL 356 to (39.39, 37.27, 0.6) mm, rotated rx 0 ry 90 rz 0 deg; joints [-9.24, 3.448, 54.52, 169.138, 58.432, -174.264]
  Call Extruder(138.299)
  MoveL 357 to (40, 37.2, 0.6) mm, rotated rx 0 ry 90 rz 0 deg; joints [-9.229, 3.494, 54.39, 169.14, 58.348, -174.251]
  Call Extruder(142.290)
  MoveL 358 to (60, 37.2, 0.6) mm, rotated rx 0 ry 90 rz 0 deg; joints [-9.027, 5.142, 49.81, 169.019, 55.449, -173.72]
  Call Extruder(142.385)
  MoveL 359 to (60.47, 37.24, 0.6) mm, rotated rx 0 ry 90 rz 0 deg; joints [-9.024, 5.185, 49.695, 169.012, 55.377, -173.705]
  Call Extruder(142.479)
  MoveL 360 to (60.93, 37.36, 0.6) mm, rotated rx 0 ry 90 rz 0 deg; joints [-9.027, 5.227, 49.58, 168.999, 55.306, -173.686]
  Call Extruder(142.573)
  MoveL 361 to (61.36, 37.55, 0.6) mm, rotated rx 0 ry 90 rz 0 deg; joints [-9.035, 5.268, 49.469, 168.98, 55.238, -173.664]
  Call Extruder(142.668)
  MoveL 362 to (61.75, 37.82, 0.6) mm, rotated rx 0 ry 90 rz 0 deg; joints [-9.048, 5.307, 49.363, 168.956, 55.174, -173.64]
  Call Extruder(142.762)
  MoveL 363 to (62.09, 38.14, 0.6) mm, rotated rx 0 ry 90 rz 0 deg; joints [-9.064, 5.342, 49.267, 168.927, 55.117, -173.614]
  Call Extruder(142.857)
  MoveL 364 to (62.38, 38.52, 0.6) mm, rotated rx 0 ry 90 rz 0 deg; joints [-9.085, 5.373, 49.184, 168.895, 55.067, -173.587]
  Call Extruder(142.951)
  MoveL 365 to (62.59, 38.94, 0.6) mm, rotated rx 0 ry 90 rz 0 deg; joints [-9.109, 5.399, 49.115, 168.86, 55.027, -173.56]
  Call Extruder(143.045)
  MoveL 366 to (62.73, 39.39, 0.6) mm, rotated rx 0 ry 90 rz 0 deg; joints [-9.136, 5.418, 49.063, 168.823, 54.998, -173.534]
  Call Extruder(143.167)
  MoveL 367 to (62.8, 40, 0.6) mm, rotated rx 0 ry 90 rz 0 deg; joints [-9.173, 5.433, 49.023, 168.775, 54.978, -173.502]
  Call Extruder(147.158)
  MoveL 368 to (62.8, 60, 0.6) mm, rotated rx 0 ry 90 rz 0 deg; joints [-10.411, 5.749, 48.173, 167.192, 54.606, -172.499]
  Call Extruder(147.253)
  MoveL 369 to (62.76, 60.47, 0.6) mm, rotated rx 0 ry 90 rz 0 deg; joints [-10.441, 5.753, 48.161, 167.155, 54.603, -172.476]
  Call Extruder(147.347)
  MoveL 370 to (62.64, 60.93, 0.6) mm, rotated rx 0 ry 90 rz 0 deg; joints [-10.47, 5.75, 48.17, 167.12, 54.612, -172.457]
  Call Extruder(147.441)
  MoveL 371 to (62.45, 61.36, 0.6) mm, rotated rx 0 ry 90 rz 0 deg; joints [-10.499, 5.739, 48.198, 167.088, 54.633, -172.441]
  Call Extruder(147.536)
  MoveL 372 to (62.18, 61.75, 0.6) mm, rotated rx 0 ry 90 rz 0 deg; joints [-10.526, 5.722, 48.245, 167.06, 54.665, -172.43]
  Call Extruder(147.630)
  MoveL 373 to (61.86, 62.1, 0.6) mm, rotated rx 0 ry 90 rz 0 deg; joints [-10.551, 5.698, 48.31, 167.036, 54.708, -172.424]
  Call Extruder(147.724)
  MoveL 374 to (61.48, 62.38, 0.6) mm, rotated rx 0 ry 90 rz 0 deg; joints [-10.573, 5.668, 48.391, 167.017, 54.76, -172.423]
  Call Extruder(147.819)
  MoveL 375 to (61.06, 62.59, 0.6) mm, rotated rx 0 ry 90 rz 0 deg; joints [-10.591, 5.633, 48.485, 167.005, 54.82, -172.426]
  Call Extruder(147.913)
  MoveL 376 to (60.61, 62.73, 0.6) mm, rotated rx 0 ry 90 rz 0 deg; joints [-10.605, 5.594, 48.589, 166.998, 54.886, -172.435]
  Call Extruder(148.035)
  MoveL 377 to (60, 62.8, 0.6) mm, rotated rx 0 ry 90 rz 0 deg; joints [-10.616, 5.54, 48.735, 166.999, 54.977, -172.452]
  Call Extruder(152.026)
  MoveL 378 to (40, 62.8, 0.6) mm, rotated rx 0 ry 90 rz 0 deg; joints [-10.853, 3.847, 53.392, 167.157, 57.896, -173.092]
  Call Extruder(152.120)
  MoveL 379 to (39.53, 62.76, 0.6) mm, rotated rx 0 ry 90 rz 0 deg; joints [-10.856, 3.809, 53.498, 167.163, 57.963, -173.108]
  Call Extruder(152.215)
  MoveL 380 to (39.07, 62.64, 0.6) mm, rotated rx 0 ry 90 rz 0 deg; joints [-10.854, 3.772, 53.604, 167.175, 58.029, -173.127]
  Call Extruder(152.309)
  MoveL 381 to (38.64, 62.45, 0.6) mm, rotated rx 0 ry 90 rz 0 deg; joints [-10.847, 3.735, 53.707, 167.192, 58.094, -173.149]
  Call Extruder(152.404)
  MoveL 382 to (38.25, 62.18, 0.6) mm, rotated rx 0 ry 90 rz 0 deg; joints [-10.835, 3.7, 53.805, 167.215, 58.154, -173.172]
  Call Extruder(152.498)
  MoveL 383 to (37.9, 61.86, 0.6) mm, rotated rx 0 ry 90 rz 0 deg; joints [-10.819, 3.669, 53.894, 167.242, 58.208, -173.197]
  Call Extruder(152.592)
  MoveL 384 to (37.62, 61.48, 0.6) mm, rotated rx 0 ry 90 rz 0 deg; joints [-10.798, 3.641, 53.972, 167.273, 58.255, -173.223]
  Call Extruder(152.687)
  MoveL 385 to (37.41, 61.06, 0.6) mm, rotated rx 0 ry 90 rz 0 deg; joints [-10.774, 3.618, 54.037, 167.307, 58.293, -173.249]
  Call Extruder(152.781)
  MoveL 386 to (37.27, 60.61, 0.6) mm, rotated rx 0 ry 90 rz 0 deg; joints [-10.747, 3.601, 54.087, 167.343, 58.321, -173.274]
  Call Extruder(152.903)
  MoveL 387 to (37.2, 60, 0.6) mm, rotated rx 0 ry 90 rz 0 deg; joints [-10.709, 3.587, 54.126, 167.39, 58.341, -173.303]
  Call Extruder(156.894)
  MoveL 388 to (37.2, 40, 0.6) mm, rotated rx 0 ry 90 rz 0 deg; joints [-9.437, 3.315, 54.899, 168.936, 58.694, -174.198]
  Call Extruder(156.988)
  MoveL 389 to (37.24, 39.53, 0.6) mm, rotated rx 0 ry 90 rz 0 deg; joints [-9.407, 3.312, 54.907, 168.972, 58.696, -174.218]
  Call Extruder(157.083)
  MoveL 390 to (37.36, 39.07, 0.6) mm, rotated rx 0 ry 90 rz 0 deg; joints [-9.376, 3.316, 54.898, 169.007, 58.687, -174.235]
  Call Extruder(157.177)
  MoveL 391 to (37.55, 38.64, 0.6) mm, rotated rx 0 ry 90 rz 0 deg; joints [-9.347, 3.325, 54.871, 169.039, 58.667, -174.249]
  Call Extruder(157.271)
  MoveL 392 to (37.82, 38.25, 0.6) mm, rotated rx 0 ry 90 rz 0 deg; joints [-9.319, 3.34, 54.828, 169.069, 58.637, -174.26]
  Call Extruder(157.366)
  MoveL 393 to (38.14, 37.91, 0.6) mm, rotated rx 0 ry 90 rz 0 deg; joints [-9.293, 3.361, 54.77, 169.094, 58.597, -174.267]
  Set speed (60.0 mm/s)
  MoveL 394 to (38.61, 38.57, 0.6) mm, rotated rx 0 ry 90 rz 0 deg; joints [-9.331, 3.404, 54.645, 169.041, 58.521, -174.226]
  Set speed (30.0 mm/s)
  Call Extruder(157.445)
  MoveL 395 to (38.92, 38.32, 0.6) mm, rotated rx 0 ry 90 rz 0 deg; joints [-9.312, 3.425, 54.586, 169.059, 58.482, -174.229]
  Call Extruder(157.525)
  MoveL 396 to (39.28, 38.14, 0.6) mm, rotated rx 0 ry 90 rz 0 deg; joints [-9.296, 3.45, 54.515, 169.071, 58.435, -174.228]
  Call Extruder(157.605)
  MoveL 397 to (39.66, 38.03, 0.6) mm, rotated rx 0 ry 90 rz 0 deg; joints [-9.285, 3.478, 54.435, 169.078, 58.383, -174.223]
  Call Extruder(157.673)
  MoveL 398 to (40, 38, 0.6) mm, rotated rx 0 ry 90 rz 0 deg; joints [-9.28, 3.504, 54.362, 169.078, 58.335, -174.216]
  Call Extruder(161.664)
  MoveL 399 to (60, 38, 0.6) mm, rotated rx 0 ry 90 rz 0 deg; joints [-9.076, 5.154, 49.78, 168.956, 55.435, -173.681]
  Call Extruder(161.744)
  MoveL 400 to (60.4, 38.04, 0.6) mm, rotated rx 0 ry 90 rz 0 deg; joints [-9.075, 5.189, 49.682, 168.949, 55.375, -173.668]
  Call Extruder(161.823)
  MoveL 401 to (60.78, 38.16, 0.6) mm, rotated rx 0 ry 90 rz 0 deg; joints [-9.079, 5.225, 49.586, 168.937, 55.315, -173.651]
  Call Extruder(161.903)
  MoveL 402 to (61.13, 38.35, 0.6) mm, rotated rx 0 ry 90 rz 0 deg; joints [-9.087, 5.259, 49.493, 168.919, 55.259, -173.632]
  Call Extruder(161.983)
  MoveL 403 to (61.43, 38.61, 0.6) mm, rotated rx 0 ry 90 rz 0 deg; joints [-9.1, 5.29, 49.41, 168.896, 55.209, -173.61]
  Call Extruder(162.062)
  MoveL 404 to (61.68, 38.92, 0.6) mm, rotated rx 0 ry 90 rz 0 deg; joints [-9.117, 5.317, 49.337, 168.87, 55.166, -173.588]
  Call Extruder(162.142)
  MoveL 405 to (61.86, 39.28, 0.6) mm, rotated rx 0 ry 90 rz 0 deg; joints [-9.137, 5.338, 49.279, 168.84, 55.132, -173.565]
  Call Extruder(162.222)
  MoveL 406 to (61.97, 39.66, 0.6) mm, rotated rx 0 ry 90 rz 0 deg; joints [-9.16, 5.353, 49.238, 168.809, 55.109, -173.543]
  Call Extruder(162.290)
  MoveL 407 to (62, 40, 0.6) mm, rotated rx 0 ry 90 rz 0 deg; joints [-9.181, 5.361, 49.218, 168.782, 55.099, -173.526]
  Call Extruder(166.281)
  MoveL 408 to (62, 60, 0.6) mm, rotated rx 0 ry 90 rz 0 deg; joints [-10.42, 5.675, 48.371, 167.201, 54.728, -172.526]
  Call Extruder(166.361)
  MoveL 409 to (61.96, 60.4, 0.6) mm, rotated rx 0 ry 90 rz 0 deg; joints [-10.445, 5.678, 48.363, 167.17, 54.726, -172.507]
  Call Extruder(166.440)
  MoveL 410 to (61.84, 60.78, 0.6) mm, rotated rx 0 ry 90 rz 0 deg; joints [-10.47, 5.674, 48.374, 167.141, 54.737, -172.492]
  Call Extruder(166.520)
  MoveL 411 to (61.65, 61.13, 0.6) mm, rotated rx 0 ry 90 rz 0 deg; joints [-10.494, 5.662, 48.406, 167.115, 54.759, -172.481]
  Call Extruder(166.600)
  MoveL 412 to (61.39, 61.44, 0.6) mm, rotated rx 0 ry 90 rz 0 deg; joints [-10.516, 5.644, 48.455, 167.093, 54.792, -172.474]
  Call Extruder(166.679)
  MoveL 413 to (61.08, 61.68, 0.6) mm, rotated rx 0 ry 90 rz 0 deg; joints [-10.535, 5.619, 48.521, 167.077, 54.835, -172.472]
  Call Extruder(166.759)
  MoveL 414 to (60.72, 61.86, 0.6) mm, rotated rx 0 ry 90 rz 0 deg; joints [-10.55, 5.59, 48.6, 167.066, 54.886, -172.475]
  Call Extruder(166.839)
  MoveL 415 to (60.34, 61.97, 0.6) mm, rotated rx 0 ry 90 rz 0 deg; joints [-10.561, 5.556, 48.69, 167.062, 54.942, -172.483]
  Call Extruder(166.907)
  MoveL 416 to (60, 62, 0.6) mm, rotated rx 0 ry 90 rz 0 deg; joints [-10.567, 5.526, 48.771, 167.063, 54.993, -172.493]
  Call Extruder(170.898)
  MoveL 417 to (40, 62, 0.6) mm, rotated rx 0 ry 90 rz 0 deg; joints [-10.802, 3.835, 53.426, 167.22, 57.911, -173.129]
  Call Extruder(170.978)
  MoveL 418 to (39.6, 61.96, 0.6) mm, rotated rx 0 ry 90 rz 0 deg; joints [-10.804, 3.803, 53.515, 167.225, 57.968, -173.143]
  Call Extruder(171.057)
  MoveL 419 to (39.22, 61.84, 0.6) mm, rotated rx 0 ry 90 rz 0 deg; joints [-10.802, 3.771, 53.605, 167.236, 58.024, -173.159]
  Call Extruder(171.137)
  MoveL 420 to (38.87, 61.65, 0.6) mm, rotated rx 0 ry 90 rz 0 deg; joints [-10.794, 3.741, 53.69, 167.253, 58.077, -173.179]
  Call Extruder(171.217)
  MoveL 421 to (38.57, 61.39, 0.6) mm, rotated rx 0 ry 90 rz 0 deg; joints [-10.781, 3.713, 53.768, 167.275, 58.124, -173.199]
  Call Extruder(171.297)
  MoveL 422 to (38.32, 61.08, 0.6) mm, rotated rx 0 ry 90 rz 0 deg; joints [-10.764, 3.689, 53.836, 167.3, 58.165, -173.221]
  Call Extruder(171.376)
  MoveL 423 to (38.14, 60.72, 0.6) mm, rotated rx 0 ry 90 rz 0 deg; joints [-10.744, 3.67, 53.891, 167.329, 58.197, -173.243]
  Call Extruder(171.456)
  MoveL 424 to (38.03, 60.34, 0.6) mm, rotated rx 0 ry 90 rz 0 deg; joints [-10.721, 3.656, 53.93, 167.359, 58.219, -173.264]
  Call Extruder(171.524)
  MoveL 425 to (38, 60, 0.6) mm, rotated rx 0 ry 90 rz 0 deg; joints [-10.7, 3.649, 53.951, 167.386, 58.23, -173.28]
  Call Extruder(175.515)
  MoveL 426 to (38, 40, 0.6) mm, rotated rx 0 ry 90 rz 0 deg; joints [-9.429, 3.376, 54.726, 168.933, 58.582, -174.178]
  Call Extruder(175.595)
  MoveL 427 to (38.04, 39.6, 0.6) mm, rotated rx 0 ry 90 rz 0 deg; joints [-9.403, 3.374, 54.731, 168.963, 58.583, -174.195]
  Call Extruder(175.675)
  MoveL 428 to (38.16, 39.22, 0.6) mm, rotated rx 0 ry 90 rz 0 deg; joints [-9.377, 3.378, 54.719, 168.992, 58.573, -174.208]
  Call Extruder(175.754)
  MoveL 429 to (38.35, 38.87, 0.6) mm, rotated rx 0 ry 90 rz 0 deg; joints [-9.353, 3.388, 54.69, 169.018, 58.552, -174.219]
  Call Extruder(175.834)
  MoveL 430 to (38.61, 38.57, 0.6) mm, rotated rx 0 ry 90 rz 0 deg; joints [-9.331, 3.404, 54.645, 169.041, 58.521, -174.226]
  Set speed (60.0 mm/s)
  MoveL 431 to (39.14, 39.16, 0.6) mm, rotated rx 0 ry 90 rz 0 deg; joints [-9.363, 3.453, 54.507, 168.993, 58.437, -174.186]
  Set speed (30.0 mm/s)
  Call Extruder(175.896)
  MoveL 432 to (39.39, 38.97, 0.6) mm, rotated rx 0 ry 90 rz 0 deg; joints [-9.348, 3.469, 54.461, 169.006, 58.406, -174.189]
  Call Extruder(175.957)
  MoveL 433 to (39.67, 38.85, 0.6) mm, rotated rx 0 ry 90 rz 0 deg; joints [-9.337, 3.489, 54.404, 169.015, 58.368, -174.187]
  Call Extruder(176.024)
  MoveL 434 to (40, 38.8, 0.6) mm, rotated rx 0 ry 90 rz 0 deg; joints [-9.331, 3.514, 54.333, 169.017, 58.322, -174.181]
  Call Extruder(180.015)
  MoveL 435 to (60, 38.8, 0.6) mm, rotated rx 0 ry 90 rz 0 deg; joints [-9.126, 5.165, 49.749, 168.893, 55.422, -173.642]
  Call Extruder(180.077)
  MoveL 436 to (60.31, 38.84, 0.6) mm, rotated rx 0 ry 90 rz 0 deg; joints [-9.126, 5.193, 49.673, 168.887, 55.375, -173.632]
  Call Extruder(180.139)
  MoveL 437 to (60.59, 38.96, 0.6) mm, rotated rx 0 ry 90 rz 0 deg; joints [-9.13, 5.22, 49.6, 168.876, 55.33, -173.618]
  Call Extruder(180.200)
  MoveL 438 to (60.84, 39.14, 0.6) mm, rotated rx 0 ry 90 rz 0 deg; joints [-9.139, 5.244, 49.533, 168.859, 55.289, -173.602]
  Call Extruder(180.262)
  MoveL 439 to (61.03, 39.39, 0.6) mm, rotated rx 0 ry 90 rz 0 deg; joints [-9.152, 5.265, 49.477, 168.838, 55.256, -173.584]
  Call Extruder(180.324)
  MoveL 440 to (61.15, 39.67, 0.6) mm, rotated rx 0 ry 90 rz 0 deg; joints [-9.169, 5.28, 49.436, 168.815, 55.233, -173.567]
  Call Extruder(180.390)
  MoveL 441 to (61.2, 40, 0.6) mm, rotated rx 0 ry 90 rz 0 deg; joints [-9.189, 5.289, 49.412, 168.789, 55.22, -173.549]
  Call Extruder(184.381)
  MoveL 442 to (61.2, 60, 0.6) mm, rotated rx 0 ry 90 rz 0 deg; joints [-10.429, 5.602, 48.568, 167.209, 54.85, -172.554]
  Call Extruder(184.443)
  MoveL 443 to (61.16, 60.31, 0.6) mm, rotated rx 0 ry 90 rz 0 deg; joints [-10.449, 5.603, 48.564, 167.185, 54.85, -172.539]
  Call Extruder(184.505)
  MoveL 444 to (61.04, 60.59, 0.6) mm, rotated rx 0 ry 90 rz 0 deg; joints [-10.468, 5.597, 48.58, 167.164, 54.862, -172.529]
  Call Extruder(184.567)
  MoveL 445 to (60.86, 60.84, 0.6) mm, rotated rx 0 ry 90 rz 0 deg; joints [-10.485, 5.584, 48.614, 167.146, 54.886, -172.522]
  Call Extruder(184.628)
  MoveL 446 to (60.61, 61.03, 0.6) mm, rotated rx 0 ry 90 rz 0 deg; joints [-10.5, 5.566, 48.665, 167.133, 54.919, -172.521]
  Call Extruder(184.690)
  MoveL 447 to (60.33, 61.15, 0.6) mm, rotated rx 0 ry 90 rz 0 deg; joints [-10.51, 5.542, 48.729, 167.127, 54.959, -172.524]
  Call Extruder(184.757)
  MoveL 448 to (60, 61.2, 0.6) mm, rotated rx 0 ry 90 rz 0 deg; joints [-10.517, 5.513, 48.808, 167.126, 55.009, -172.533]
  Call Extruder(188.748)
  MoveL 449 to (40, 61.2, 0.6) mm, rotated rx 0 ry 90 rz 0 deg; joints [-10.752, 3.823, 53.459, 167.282, 57.926, -173.166]
  Call Extruder(188.810)
  MoveL 450 to (39.69, 61.16, 0.6) mm, rotated rx 0 ry 90 rz 0 deg; joints [-10.753, 3.798, 53.529, 167.287, 57.97, -173.177]
  Call Extruder(188.871)
  MoveL 451 to (39.41, 61.04, 0.6) mm, rotated rx 0 ry 90 rz 0 deg; joints [-10.749, 3.774, 53.597, 167.297, 58.013, -173.191]
  Call Extruder(188.933)
  MoveL 452 to (39.16, 60.86, 0.6) mm, rotated rx 0 ry 90 rz 0 deg; joints [-10.74, 3.752, 53.66, 167.313, 58.051, -173.207]
  Call Extruder(188.995)
  MoveL 453 to (38.97, 60.61, 0.6) mm, rotated rx 0 ry 90 rz 0 deg; joints [-10.727, 3.733, 53.712, 167.333, 58.082, -173.223]
  Call Extruder(189.056)
  MoveL 454 to (38.85, 60.33, 0.6) mm, rotated rx 0 ry 90 rz 0 deg; joints [-10.711, 3.72, 53.751, 167.356, 58.105, -173.24]
  Call Extruder(189.123)
  MoveL 455 to (38.8, 60, 0.6) mm, rotated rx 0 ry 90 rz 0 deg; joints [-10.69, 3.711, 53.775, 167.382, 58.118, -173.257]
  Call Extruder(193.114)
  MoveL 456 to (38.8, 40, 0.6) mm, rotated rx 0 ry 90 rz 0 deg; joints [-9.42, 3.437, 54.552, 168.929, 58.471, -174.158]
  Call Extruder(193.176)
  MoveL 457 to (38.84, 39.69, 0.6) mm, rotated rx 0 ry 90 rz 0 deg; joints [-9.4, 3.436, 54.554, 168.953, 58.47, -174.17]
  Call Extruder(193.238)
  MoveL 458 to (38.96, 39.41, 0.6) mm, rotated rx 0 ry 90 rz 0 deg; joints [-9.381, 3.442, 54.539, 168.974, 58.458, -174.18]
  Call Extruder(193.299)
  MoveL 459 to (39.14, 39.16, 0.6) mm, rotated rx 0 ry 90 rz 0 deg; joints [-9.363, 3.453, 54.507, 168.993, 58.437, -174.186]
  Set speed (60.0 mm/s)
  MoveL 460 to (39.75, 39.69, 0.6) mm, rotated rx 0 ry 90 rz 0 deg; joints [-9.39, 3.506, 54.356, 168.949, 58.343, -174.148]
  Set speed (30.0 mm/s)
  Call Extruder(193.335)
  MoveL 461 to (39.91, 39.61, 0.6) mm, rotated rx 0 ry 90 rz 0 deg; joints [-9.384, 3.517, 54.324, 168.955, 58.322, -174.147]
  Call Extruder(193.353)
  MoveL 462 to (40, 39.6, 0.6) mm, rotated rx 0 ry 90 rz 0 deg; joints [-9.382, 3.524, 54.304, 168.955, 58.309, -174.145]
  Call Extruder(197.344)
  MoveL 463 to (60, 39.6, 0.6) mm, rotated rx 0 ry 90 rz 0 deg; joints [-9.176, 5.176, 49.718, 168.83, 55.408, -173.604]
  Call Extruder(197.379)
  MoveL 464 to (60.17, 39.64, 0.6) mm, rotated rx 0 ry 90 rz 0 deg; joints [-9.177, 5.192, 49.674, 168.826, 55.381, -173.597]
  Call Extruder(197.415)
  MoveL 465 to (60.31, 39.75, 0.6) mm, rotated rx 0 ry 90 rz 0 deg; joints [-9.182, 5.206, 49.637, 168.816, 55.358, -173.587]
  Call Extruder(197.450)
  MoveL 466 to (60.39, 39.91, 0.6) mm, rotated rx 0 ry 90 rz 0 deg; joints [-9.192, 5.215, 49.612, 168.803, 55.344, -173.577]
  Call Extruder(197.468)
  MoveL 467 to (60.4, 40, 0.6) mm, rotated rx 0 ry 90 rz 0 deg; joints [-9.197, 5.218, 49.606, 168.795, 55.341, -173.573]
  Call Extruder(201.460)
  MoveL 468 to (60.4, 60, 0.6) mm, rotated rx 0 ry 90 rz 0 deg; joints [-10.438, 5.529, 48.764, 167.217, 54.972, -172.581]
  Call Extruder(201.495)
  MoveL 469 to (60.36, 60.17, 0.6) mm, rotated rx 0 ry 90 rz 0 deg; joints [-10.449, 5.528, 48.766, 167.204, 54.974, -172.573]
  Call Extruder(201.531)
  MoveL 470 to (60.25, 60.31, 0.6) mm, rotated rx 0 ry 90 rz 0 deg; joints [-10.459, 5.52, 48.787, 167.194, 54.988, -172.57]
  Call Extruder(201.566)
  MoveL 471 to (60.09, 60.39, 0.6) mm, rotated rx 0 ry 90 rz 0 deg; joints [-10.466, 5.507, 48.823, 167.19, 55.011, -172.571]
  Call Extruder(201.584)
  MoveL 472 to (60, 60.4, 0.6) mm, rotated rx 0 ry 90 rz 0 deg; joints [-10.468, 5.499, 48.844, 167.19, 55.024, -172.574]
  Call Extruder(205.575)
  MoveL 473 to (40, 60.4, 0.6) mm, rotated rx 0 ry 90 rz 0 deg; joints [-10.701, 3.811, 53.493, 167.344, 57.941, -173.203]
  Call Extruder(205.611)
  MoveL 474 to (39.83, 60.36, 0.6) mm, rotated rx 0 ry 90 rz 0 deg; joints [-10.701, 3.797, 53.533, 167.348, 57.966, -173.21]
  Call Extruder(205.646)
  MoveL 475 to (39.69, 60.25, 0.6) mm, rotated rx 0 ry 90 rz 0 deg; joints [-10.695, 3.784, 53.568, 167.357, 57.988, -173.219]
  Call Extruder(205.682)
  MoveL 476 to (39.61, 60.09, 0.6) mm, rotated rx 0 ry 90 rz 0 deg; joints [-10.686, 3.776, 53.592, 167.37, 58.002, -173.229]
  Call Extruder(205.700)
  MoveL 477 to (39.6, 60, 0.6) mm, rotated rx 0 ry 90 rz 0 deg; joints [-10.681, 3.774, 53.598, 167.377, 58.005, -173.233]
  Call Extruder(209.691)
  MoveL 478 to (39.6, 40, 0.6) mm, rotated rx 0 ry 90 rz 0 deg; joints [-9.412, 3.498, 54.377, 168.926, 58.359, -174.138]
  Call Extruder(209.726)
  MoveL 479 to (39.64, 39.83, 0.6) mm, rotated rx 0 ry 90 rz 0 deg; joints [-9.4, 3.499, 54.375, 168.939, 58.356, -174.144]
  Call Extruder(209.762)
  MoveL 480 to (39.75, 39.69, 0.6) mm, rotated rx 0 ry 90 rz 0 deg; joints [-9.39, 3.506, 54.356, 168.949, 58.343, -174.148]
  Call Extruder(209.162)
  MoveL 481 to (39.75, 39.69, 0.6) mm, rotated rx 0 ry 90 rz 0 deg; joints [-9.39, 3.506, 54.356, 168.949, 58.343, -174.148]
  Set speed (60.0 mm/s)
  MoveL 482 to (40.5, 59.53, 0.6) mm, rotated rx 0 ry 90 rz 0 deg; joints [-10.64, 3.838, 53.418, 167.409, 57.887, -173.228]
  Set speed (1000.0 mm/s)
  MoveL 483 to (40.4, 59.6, 0.6) mm, rotated rx 0 ry 90 rz 0 deg; joints [-10.646, 3.831, 53.438, 167.404, 57.9, -173.228]
  Set speed (30.0 mm/s)
  Call Extruder(209.762)
  MoveL 484 to (40.4, 59.6, 0.6) mm, rotated rx 0 ry 90 rz 0 deg; joints [-10.646, 3.831, 53.438, 167.404, 57.9, -173.228]
  Call Extruder(213.593)
  MoveL 485 to (40.4, 40.4, 0.6) mm, rotated rx 0 ry 90 rz 0 deg; joints [-9.429, 3.565, 54.188, 168.891, 58.24, -174.099]
  Call Extruder(217.425)
  MoveL 486 to (59.6, 40.4, 0.6) mm, rotated rx 0 ry 90 rz 0 deg; joints [-9.23, 5.152, 49.783, 168.771, 55.454, -173.576]
  Call Extruder(221.257)
  MoveL 487 to (59.6, 59.6, 0.6) mm, rotated rx 0 ry 90 rz 0 deg; joints [-10.423, 5.45, 48.978, 167.257, 55.101, -172.628]
  Call Extruder(225.088)
  MoveL 488 to (40.4, 59.6, 0.6) mm, rotated rx 0 ry 90 rz 0 deg; joints [-10.646, 3.831, 53.438, 167.404, 57.9, -173.228]
  Set speed (60.0 mm/s)
  MoveL 489 to (40.4, 59.2, 0.6) mm, rotated rx 0 ry 90 rz 0 deg; joints [-10.621, 3.825, 53.454, 167.435, 57.908, -173.247]
  Set speed (1000.0 mm/s)
  MoveL 490 to (41.19, 58.81, 0.6) mm, rotated rx 0 ry 90 rz 0 deg; joints [-10.587, 3.881, 53.295, 167.461, 57.803, -173.242]
  Set speed (30.0 mm/s)
  Call Extruder(228.604)
  MoveL 491 to (41.19, 41.19, 0.6) mm, rotated rx 0 ry 90 rz 0 deg; joints [-9.471, 3.637, 53.985, 168.827, 58.116, -174.044]
  Call Extruder(232.121)
  MoveL 492 to (58.81, 41.19, 0.6) mm, rotated rx 0 ry 90 rz 0 deg; joints [-9.287, 5.094, 49.941, 168.715, 55.559, -173.561]
  Call Extruder(235.637)
  MoveL 493 to (58.81, 58.81, 0.6) mm, rotated rx 0 ry 90 rz 0 deg; joints [-10.383, 5.365, 49.205, 167.327, 55.235, -172.694]
  Call Extruder(239.153)
  MoveL 494 to (41.19, 58.81, 0.6) mm, rotated rx 0 ry 90 rz 0 deg; joints [-10.587, 3.881, 53.295, 167.461, 57.803, -173.242]
  Set speed (60.0 mm/s)
  MoveL 495 to (42.61, 58.45, 0.6) mm, rotated rx 0 ry 90 rz 0 deg; joints [-10.547, 3.989, 52.993, 167.48, 57.609, -173.216]
  Set speed (30.0 mm/s)
  Call Extruder(239.453)
  MoveL 496 to (41.55, 57.39, 0.6) mm, rotated rx 0 ry 90 rz 0 deg; joints [-10.493, 3.889, 53.274, 167.569, 57.779, -173.297]
  Set speed (60.0 mm/s)
  MoveL 497 to (41.55, 56.26, 0.6) mm, rotated rx 0 ry 90 rz 0 deg; joints [-10.421, 3.872, 53.321, 167.657, 57.8, -173.349]
  Set speed (30.0 mm/s)
  Call Extruder(240.071)
  MoveL 498 to (43.74, 58.45, 0.6) mm, rotated rx 0 ry 90 rz 0 deg; joints [-10.534, 4.08, 52.739, 167.474, 57.448, -173.183]
  Set speed (60.0 mm/s)
  MoveL 499 to (44.87, 58.45, 0.6) mm, rotated rx 0 ry 90 rz 0 deg; joints [-10.521, 4.171, 52.484, 167.466, 57.287, -173.149]
  Set speed (30.0 mm/s)
  Call Extruder(241.009)
  MoveL 500 to (41.55, 55.13, 0.6) mm, rotated rx 0 ry 90 rz 0 deg; joints [-10.35, 3.856, 53.367, 167.745, 57.821, -173.401]
  Set speed (60.0 mm/s)
  MoveL 501 to (41.55, 53.99, 0.6) mm, rotated rx 0 ry 90 rz 0 deg; joints [-10.278, 3.84, 53.412, 167.833, 57.841, -173.453]
  Set speed (30.0 mm/s)
  Call Extruder(242.266)
  MoveL 502 to (46, 58.45, 0.6) mm, rotated rx 0 ry 90 rz 0 deg; joints [-10.508, 4.263, 52.227, 167.459, 57.124, -173.115]
  Set speed (60.0 mm/s)
  MoveL 503 to (47.14, 58.45, 0.6) mm, rotated rx 0 ry 90 rz 0 deg; joints [-10.494, 4.356, 51.969, 167.451, 56.962, -173.081]
  Set speed (30.0 mm/s)
  Call Extruder(243.843)
  MoveL 504 to (41.55, 52.86, 0.6) mm, rotated rx 0 ry 90 rz 0 deg; joints [-10.207, 3.824, 53.458, 167.921, 57.862, -173.505]
  Set speed (60.0 mm/s)
  MoveL 505 to (41.55, 51.73, 0.6) mm, rotated rx 0 ry 90 rz 0 deg; joints [-10.135, 3.807, 53.503, 168.008, 57.882, -173.557]
  Set speed (30.0 mm/s)
  Call Extruder(245.739)
  MoveL 506 to (48.27, 58.45, 0.6) mm, rotated rx 0 ry 90 rz 0 deg; joints [-10.481, 4.45, 51.71, 167.443, 56.798, -173.046]
  Set speed (60.0 mm/s)
  MoveL 507 to (49.4, 58.45, 0.6) mm, rotated rx 0 ry 90 rz 0 deg; joints [-10.468, 4.544, 51.449, 167.435, 56.634, -173.011]
  Set speed (30.0 mm/s)
  Call Extruder(247.954)
  MoveL 508 to (41.55, 50.6, 0.6) mm, rotated rx 0 ry 90 rz 0 deg; joints [-10.064, 3.792, 53.548, 168.096, 57.903, -173.609]
  Set speed (60.0 mm/s)
  MoveL 509 to (41.55, 49.47, 0.6) mm, rotated rx 0 ry 90 rz 0 deg; joints [-9.992, 3.776, 53.592, 168.184, 57.923, -173.66]
  Set speed (30.0 mm/s)
  Call Extruder(250.488)
  MoveL 510 to (50.53, 58.45, 0.6) mm, rotated rx 0 ry 90 rz 0 deg; joints [-10.455, 4.639, 51.187, 167.427, 56.469, -172.976]
  Set speed (60.0 mm/s)
  MoveL 511 to (51.66, 58.45, 0.6) mm, rotated rx 0 ry 90 rz 0 deg; joints [-10.442, 4.735, 50.923, 167.418, 56.304, -172.941]
  Set speed (30.0 mm/s)
  Call Extruder(253.342)
  MoveL 512 to (41.55, 48.34, 0.6) mm, rotated rx 0 ry 90 rz 0 deg; joints [-9.92, 3.76, 53.636, 168.272, 57.943, -173.712]
  Set speed (60.0 mm/s)
  MoveL 513 to (41.55, 47.21, 0.6) mm, rotated rx 0 ry 90 rz 0 deg; joints [-9.849, 3.745, 53.68, 168.359, 57.962, -173.763]
  Set speed (30.0 mm/s)
  Call Extruder(256.515)
  MoveL 514 to (52.79, 58.45, 0.6) mm, rotated rx 0 ry 90 rz 0 deg; joints [-10.429, 4.832, 50.658, 167.409, 56.138, -172.906]
  Set speed (60.0 mm/s)
  MoveL 515 to (53.92, 58.45, 0.6) mm, rotated rx 0 ry 90 rz 0 deg; joints [-10.416, 4.929, 50.391, 167.399, 55.971, -172.87]
  Set speed (30.0 mm/s)
  Call Extruder(260.007)
  MoveL 516 to (41.55, 46.07, 0.6) mm, rotated rx 0 ry 90 rz 0 deg; joints [-9.777, 3.729, 53.723, 168.447, 57.982, -173.814]
  Set speed (60.0 mm/s)
  MoveL 517 to (41.55, 44.94, 0.6) mm, rotated rx 0 ry 90 rz 0 deg; joints [-9.705, 3.714, 53.766, 168.534, 58.001, -173.866]
  Set speed (30.0 mm/s)
  Call Extruder(263.819)
  MoveL 518 to (55.05, 58.45, 0.6) mm, rotated rx 0 ry 90 rz 0 deg; joints [-10.403, 5.028, 50.123, 167.39, 55.804, -172.834]
  Set speed (60.0 mm/s)
  MoveL 519 to (56.19, 58.45, 0.6) mm, rotated rx 0 ry 90 rz 0 deg; joints [-10.39, 5.127, 49.853, 167.38, 55.635, -172.797]
  Set speed (30.0 mm/s)
  Call Extruder(267.950)
  MoveL 520 to (41.55, 43.81, 0.6) mm, rotated rx 0 ry 90 rz 0 deg; joints [-9.633, 3.699, 53.808, 168.622, 58.021, -173.917]
  Set speed (60.0 mm/s)
  MoveL 521 to (41.55, 42.68, 0.6) mm, rotated rx 0 ry 90 rz 0 deg; joints [-9.561, 3.684, 53.851, 168.71, 58.04, -173.967]
  Set speed (30.0 mm/s)
  Call Extruder(272.400)
  MoveL 522 to (57.32, 58.45, 0.6) mm, rotated rx 0 ry 90 rz 0 deg; joints [-10.377, 5.226, 49.581, 167.37, 55.466, -172.76]
  Set speed (60.0 mm/s)
  MoveL 523 to (58.45, 58.45, 0.6) mm, rotated rx 0 ry 90 rz 0 deg; joints [-10.364, 5.327, 49.309, 167.359, 55.297, -172.724]
  Set speed (30.0 mm/s)
  Call Extruder(277.170)
  MoveL 524 to (41.55, 41.55, 0.6) mm, rotated rx 0 ry 90 rz 0 deg; joints [-9.49, 3.669, 53.893, 168.797, 58.059, -174.018]
  Set speed (60.0 mm/s)
  MoveL 525 to (42.68, 41.55, 0.6) mm, rotated rx 0 ry 90 rz 0 deg; joints [-9.478, 3.758, 53.642, 168.791, 57.899, -173.989]
  Set speed (30.0 mm/s)
  Call Extruder(281.620)
  MoveL 526 to (58.45, 57.32, 0.6) mm, rotated rx 0 ry 90 rz 0 deg; joints [-10.294, 5.309, 49.358, 167.449, 55.318, -172.78]
  Set speed (60.0 mm/s)
  MoveL 527 to (58.45, 56.19, 0.6) mm, rotated rx 0 ry 90 rz 0 deg; joints [-10.224, 5.29, 49.408, 167.538, 55.34, -172.836]
  Set speed (30.0 mm/s)
  Call Extruder(285.751)
  MoveL 528 to (43.81, 41.55, 0.6) mm, rotated rx 0 ry 90 rz 0 deg; joints [-9.466, 3.847, 53.391, 168.786, 57.739, -173.959]
  Set speed (60.0 mm/s)
  MoveL 529 to (44.94, 41.55, 0.6) mm, rotated rx 0 ry 90 rz 0 deg; joints [-9.454, 3.937, 53.138, 168.78, 57.578, -173.929]
  Set speed (30.0 mm/s)
  Call Extruder(289.563)
  MoveL 530 to (58.45, 55.06, 0.6) mm, rotated rx 0 ry 90 rz 0 deg; joints [-10.154, 5.272, 49.457, 167.627, 55.362, -172.893]
  Set speed (60.0 mm/s)
  MoveL 531 to (58.45, 53.92, 0.6) mm, rotated rx 0 ry 90 rz 0 deg; joints [-10.084, 5.254, 49.506, 167.716, 55.383, -172.949]
  Set speed (30.0 mm/s)
  Call Extruder(293.055)
  MoveL 532 to (46.08, 41.55, 0.6) mm, rotated rx 0 ry 90 rz 0 deg; joints [-9.442, 4.028, 52.884, 168.773, 57.416, -173.899]
  Set speed (60.0 mm/s)
  MoveL 533 to (47.21, 41.55, 0.6) mm, rotated rx 0 ry 90 rz 0 deg; joints [-9.43, 4.119, 52.628, 168.767, 57.254, -173.868]
  Set speed (30.0 mm/s)
  Call Extruder(296.228)
  MoveL 534 to (58.45, 52.79, 0.6) mm, rotated rx 0 ry 90 rz 0 deg; joints [-10.013, 5.237, 49.554, 167.806, 55.404, -173.005]
  Set speed (60.0 mm/s)
  MoveL 535 to (58.45, 51.66, 0.6) mm, rotated rx 0 ry 90 rz 0 deg; joints [-9.943, 5.219, 49.602, 167.895, 55.425, -173.061]
  Set speed (30.0 mm/s)
  Call Extruder(299.082)
  MoveL 536 to (48.34, 41.55, 0.6) mm, rotated rx 0 ry 90 rz 0 deg; joints [-9.418, 4.211, 52.372, 168.76, 57.091, -173.838]
  Set speed (60.0 mm/s)
  MoveL 537 to (49.47, 41.55, 0.6) mm, rotated rx 0 ry 90 rz 0 deg; joints [-9.406, 4.304, 52.114, 168.753, 56.928, -173.807]
  Set speed (30.0 mm/s)
  Call Extruder(301.616)
  MoveL 538 to (58.45, 50.53, 0.6) mm, rotated rx 0 ry 90 rz 0 deg; joints [-9.873, 5.201, 49.65, 167.984, 55.446, -173.116]
  Set speed (60.0 mm/s)
  MoveL 539 to (58.45, 49.4, 0.6) mm, rotated rx 0 ry 90 rz 0 deg; joints [-9.802, 5.184, 49.697, 168.073, 55.467, -173.172]
  Set speed (30.0 mm/s)
  Call Extruder(303.831)
  MoveL 540 to (50.6, 41.55, 0.6) mm, rotated rx 0 ry 90 rz 0 deg; joints [-9.394, 4.398, 51.854, 168.746, 56.764, -173.776]
  Set speed (60.0 mm/s)
  MoveL 541 to (51.73, 41.55, 0.6) mm, rotated rx 0 ry 90 rz 0 deg; joints [-9.383, 4.492, 51.593, 168.739, 56.599, -173.745]
  Set speed (30.0 mm/s)
  Call Extruder(305.727)
  MoveL 542 to (58.45, 48.27, 0.6) mm, rotated rx 0 ry 90 rz 0 deg; joints [-9.732, 5.167, 49.744, 168.162, 55.488, -173.227]
  Set speed (60.0 mm/s)
  MoveL 543 to (58.45, 47.14, 0.6) mm, rotated rx 0 ry 90 rz 0 deg; joints [-9.662, 5.15, 49.79, 168.251, 55.508, -173.283]
  Set speed (30.0 mm/s)
  Call Extruder(307.304)
  MoveL 544 to (52.86, 41.55, 0.6) mm, rotated rx 0 ry 90 rz 0 deg; joints [-9.371, 4.587, 51.331, 168.731, 56.434, -173.713]
  Set speed (60.0 mm/s)
  MoveL 545 to (53.99, 41.55, 0.6) mm, rotated rx 0 ry 90 rz 0 deg; joints [-9.359, 4.683, 51.067, 168.723, 56.268, -173.682]
  Set speed (30.0 mm/s)
  Call Extruder(308.561)
  MoveL 546 to (58.45, 46, 0.6) mm, rotated rx 0 ry 90 rz 0 deg; joints [-9.591, 5.133, 49.836, 168.34, 55.528, -173.338]
  Set speed (60.0 mm/s)
  MoveL 547 to (58.45, 44.87, 0.6) mm, rotated rx 0 ry 90 rz 0 deg; joints [-9.521, 5.116, 49.882, 168.429, 55.549, -173.393]
  Set speed (30.0 mm/s)
  Call Extruder(309.499)
  MoveL 548 to (55.13, 41.55, 0.6) mm, rotated rx 0 ry 90 rz 0 deg; joints [-9.348, 4.779, 50.802, 168.715, 56.101, -173.65]
  Set speed (60.0 mm/s)
  MoveL 549 to (56.26, 41.55, 0.6) mm, rotated rx 0 ry 90 rz 0 deg; joints [-9.336, 4.877, 50.535, 168.707, 55.933, -173.617]
  Set speed (30.0 mm/s)
  Call Extruder(310.118)
  MoveL 550 to (58.45, 43.74, 0.6) mm, rotated rx 0 ry 90 rz 0 deg; joints [-9.45, 5.099, 49.927, 168.518, 55.569, -173.448]
  Set speed (60.0 mm/s)
  MoveL 551 to (58.45, 42.61, 0.6) mm, rotated rx 0 ry 90 rz 0 deg; joints [-9.38, 5.083, 49.972, 168.607, 55.588, -173.503]
  Set speed (30.0 mm/s)
  Call Extruder(310.417)
  MoveL 552 to (57.39, 41.55, 0.6) mm, rotated rx 0 ry 90 rz 0 deg; joints [-9.324, 4.975, 50.267, 168.698, 55.765, -173.585]
  Set speed (60.0 mm/s)
  MoveL 553 to (40.47, 59.53, 0.6) mm, rotated rx 0 ry 90 rz 0 deg; joints [-10.641, 3.835, 53.425, 167.409, 57.891, -173.229]
  Set speed (1000.0 mm/s)
  MoveL 554 to (40.4, 59.6, 0.6) mm, rotated rx 0 ry 90 rz 0 deg; joints [-10.646, 3.831, 53.438, 167.404, 57.9, -173.228]
  Call M_RunCode(106,0)
  Set speed (90.0 mm/s)
  MoveL 555 to (40.4, 59.6, 1) mm, rotated rx 0 ry 90 rz 0 deg; joints [-10.646, 3.788, 53.485, 167.404, 57.904, -173.229]
  Set speed (30.0 mm/s)
  Call Extruder(312.971)
  MoveL 556 to (40.4, 40.4, 1) mm, rotated rx 0 ry 90 rz 0 deg; joints [-9.429, 3.522, 54.234, 168.892, 58.243, -174.1]
  Call Extruder(315.526)
  MoveL 557 to (59.6, 40.4, 1) mm, rotated rx 0 ry 90 rz 0 deg; joints [-9.23, 5.108, 49.833, 168.771, 55.46, -173.578]
  Call Extruder(318.080)
  MoveL 558 to (59.6, 59.6, 1) mm, rotated rx 0 ry 90 rz 0 deg; joints [-10.423, 5.405, 49.028, 167.258, 55.106, -172.629]
  Call Extruder(320.634)
  MoveL 559 to (40.4, 59.6, 1) mm, rotated rx 0 ry 90 rz 0 deg; joints [-10.646, 3.788, 53.485, 167.404, 57.904, -173.229]
  Set speed (90.0 mm/s)
  MoveL 560 to (40.4, 59.2, 1) mm, rotated rx 0 ry 90 rz 0 deg; joints [-10.621, 3.782, 53.501, 167.435, 57.911, -173.248]
  Set speed (1000.0 mm/s)
  MoveL 561 to (41.19, 58.81, 1) mm, rotated rx 0 ry 90 rz 0 deg; joints [-10.587, 3.838, 53.342, 167.461, 57.807, -173.243]
  Set speed (30.0 mm/s)
  Call Extruder(322.979)
  MoveL 562 to (41.19, 41.19, 1) mm, rotated rx 0 ry 90 rz 0 deg; joints [-9.471, 3.594, 54.032, 168.827, 58.119, -174.045]
  Call Extruder(325.323)
  MoveL 563 to (58.81, 41.19, 1) mm, rotated rx 0 ry 90 rz 0 deg; joints [-9.287, 5.05, 49.991, 168.716, 55.564, -173.562]
  Call Extruder(327.667)
  MoveL 564 to (58.81, 58.81, 1) mm, rotated rx 0 ry 90 rz 0 deg; joints [-10.383, 5.321, 49.255, 167.328, 55.241, -172.695]
  Call Extruder(330.011)
  MoveL 565 to (41.19, 58.81, 1) mm, rotated rx 0 ry 90 rz 0 deg; joints [-10.587, 3.838, 53.342, 167.461, 57.807, -173.243]
  Set speed (90.0 mm/s)
  MoveL 566 to (41.55, 42.17, 1) mm, rotated rx 0 ry 90 rz 0 deg; joints [-9.529, 3.635, 53.916, 168.749, 58.052, -173.991]
  Set speed (30.0 mm/s)
  Call Extruder(330.128)
  MoveL 567 to (42.17, 41.55, 1) mm, rotated rx 0 ry 90 rz 0 deg; joints [-9.483, 3.675, 53.802, 168.794, 57.975, -174.003]
  Set speed (90.0 mm/s)
  MoveL 568 to (43.3, 41.55, 1) mm, rotated rx 0 ry 90 rz 0 deg; joints [-9.471, 3.764, 53.551, 168.789, 57.815, -173.973]
  Set speed (30.0 mm/s)
  Call Extruder(330.458)
  MoveL 569 to (41.55, 43.3, 1) mm, rotated rx 0 ry 90 rz 0 deg; joints [-9.601, 3.649, 53.874, 168.662, 58.033, -173.94]
  Set speed (90.0 mm/s)
  MoveL 570 to (41.55, 44.43, 1) mm, rotated rx 0 ry 90 rz 0 deg; joints [-9.673, 3.664, 53.832, 168.574, 58.014, -173.889]
  Set speed (30.0 mm/s)
  Call Extruder(331.001)
  MoveL 571 to (44.43, 41.55, 1) mm, rotated rx 0 ry 90 rz 0 deg; joints [-9.459, 3.854, 53.299, 168.783, 57.654, -173.943]
  Set speed (90.0 mm/s)
  MoveL 572 to (45.57, 41.55, 1) mm, rotated rx 0 ry 90 rz 0 deg; joints [-9.447, 3.944, 53.046, 168.777, 57.493, -173.913]
  Set speed (30.0 mm/s)
  Call Extruder(331.757)
  MoveL 573 to (41.55, 45.57, 1) mm, rotated rx 0 ry 90 rz 0 deg; joints [-9.745, 3.68, 53.789, 168.487, 57.994, -173.838]
  Set speed (90.0 mm/s)
  MoveL 574 to (41.55, 46.7, 1) mm, rotated rx 0 ry 90 rz 0 deg; joints [-9.816, 3.695, 53.746, 168.399, 57.975, -173.787]
  Set speed (30.0 mm/s)
  Call Extruder(332.725)
  MoveL 575 to (46.7, 41.55, 1) mm, rotated rx 0 ry 90 rz 0 deg; joints [-9.435, 4.035, 52.791, 168.77, 57.331, -173.883]
  Set speed (90.0 mm/s)
  MoveL 576 to (47.83, 41.55, 1) mm, rotated rx 0 ry 90 rz 0 deg; joints [-9.423, 4.126, 52.535, 168.764, 57.169, -173.853]
  Set speed (30.0 mm/s)
  Call Extruder(333.907)
  MoveL 577 to (41.55, 47.83, 1) mm, rotated rx 0 ry 90 rz 0 deg; joints [-9.888, 3.71, 53.703, 168.312, 57.955, -173.736]
  Set speed (90.0 mm/s)
  MoveL 578 to (41.55, 48.96, 1) mm, rotated rx 0 ry 90 rz 0 deg; joints [-9.96, 3.726, 53.659, 168.224, 57.935, -173.684]
  Set speed (30.0 mm/s)
  Call Extruder(335.301)
  MoveL 579 to (48.96, 41.55, 1) mm, rotated rx 0 ry 90 rz 0 deg; joints [-9.412, 4.219, 52.278, 168.757, 57.006, -173.822]
  Set speed (90.0 mm/s)
  MoveL 580 to (50.09, 41.55, 1) mm, rotated rx 0 ry 90 rz 0 deg; joints [-9.4, 4.312, 52.019, 168.75, 56.842, -173.791]
  Set speed (30.0 mm/s)
  Call Extruder(336.908)
  MoveL 581 to (41.55, 50.09, 1) mm, rotated rx 0 ry 90 rz 0 deg; joints [-10.031, 3.741, 53.615, 168.136, 57.915, -173.633]
  Set speed (90.0 mm/s)
  MoveL 582 to (41.55, 51.22, 1) mm, rotated rx 0 ry 90 rz 0 deg; joints [-10.103, 3.757, 53.57, 168.048, 57.895, -173.581]
  Set speed (30.0 mm/s)
  Call Extruder(338.728)
  MoveL 583 to (51.22, 41.55, 1) mm, rotated rx 0 ry 90 rz 0 deg; joints [-9.388, 4.406, 51.759, 168.743, 56.678, -173.76]
  Set speed (90.0 mm/s)
  MoveL 584 to (52.35, 41.55, 1) mm, rotated rx 0 ry 90 rz 0 deg; joints [-9.376, 4.5, 51.497, 168.735, 56.513, -173.729]
  Set speed (30.0 mm/s)
  Call Extruder(340.761)
  MoveL 585 to (41.55, 52.35, 1) mm, rotated rx 0 ry 90 rz 0 deg; joints [-10.175, 3.773, 53.525, 167.961, 57.875, -173.53]
  Set speed (90.0 mm/s)
  MoveL 586 to (41.55, 53.48, 1) mm, rotated rx 0 ry 90 rz 0 deg; joints [-10.246, 3.789, 53.48, 167.873, 57.855, -173.478]
  Set speed (30.0 mm/s)
  Call Extruder(343.007)
  MoveL 587 to (53.48, 41.55, 1) mm, rotated rx 0 ry 90 rz 0 deg; joints [-9.365, 4.596, 51.235, 168.728, 56.347, -173.697]
  Set speed (90.0 mm/s)
  MoveL 588 to (54.62, 41.55, 1) mm, rotated rx 0 ry 90 rz 0 deg; joints [-9.353, 4.692, 50.97, 168.72, 56.181, -173.665]
  Set speed (30.0 mm/s)
  Call Extruder(345.465)
  MoveL 589 to (41.55, 54.62, 1) mm, rotated rx 0 ry 90 rz 0 deg; joints [-10.318, 3.805, 53.434, 167.785, 57.834, -173.426]
  Set speed (90.0 mm/s)
  MoveL 590 to (41.55, 55.75, 1) mm, rotated rx 0 ry 90 rz 0 deg; joints [-10.389, 3.822, 53.388, 167.697, 57.813, -173.374]
  Set speed (30.0 mm/s)
  Call Extruder(348.137)
  MoveL 591 to (55.75, 41.55, 1) mm, rotated rx 0 ry 90 rz 0 deg; joints [-9.341, 4.789, 50.704, 168.711, 56.014, -173.633]
  Set speed (90.0 mm/s)
  MoveL 592 to (56.88, 41.55, 1) mm, rotated rx 0 ry 90 rz 0 deg; joints [-9.33, 4.886, 50.437, 168.703, 55.846, -173.601]
  Set speed (30.0 mm/s)
  Call Extruder(351.021)
  MoveL 593 to (41.55, 56.88, 1) mm, rotated rx 0 ry 90 rz 0 deg; joints [-10.461, 3.838, 53.342, 167.609, 57.792, -173.321]
  Set speed (90.0 mm/s)
  MoveL 594 to (41.55, 58.01, 1) mm, rotated rx 0 ry 90 rz 0 deg; joints [-10.532, 3.855, 53.295, 167.521, 57.771, -173.269]
  Set speed (30.0 mm/s)
  Call Extruder(354.118)
  MoveL 595 to (58.01, 41.55, 1) mm, rotated rx 0 ry 90 rz 0 deg; joints [-9.318, 4.985, 50.168, 168.694, 55.678, -173.568]
  Set speed (90.0 mm/s)
  MoveL 596 to (58.45, 42.24, 1) mm, rotated rx 0 ry 90 rz 0 deg; joints [-9.357, 5.033, 50.036, 168.636, 55.6, -173.522]
  Set speed (30.0 mm/s)
  Call Extruder(357.168)
  MoveL 597 to (42.24, 58.45, 1) mm, rotated rx 0 ry 90 rz 0 deg; joints [-10.552, 3.916, 53.123, 167.483, 57.665, -173.228]
  Set speed (90.0 mm/s)
  MoveL 598 to (43.37, 58.45, 1) mm, rotated rx 0 ry 90 rz 0 deg; joints [-10.538, 4.007, 52.869, 167.476, 57.505, -173.195]
  Set speed (30.0 mm/s)
  Call Extruder(360.004)
  MoveL 599 to (58.45, 43.37, 1) mm, rotated rx 0 ry 90 rz 0 deg; joints [-9.427, 5.05, 49.991, 168.547, 55.58, -173.467]
  Set speed (90.0 mm/s)
  MoveL 600 to (58.45, 44.51, 1) mm, rotated rx 0 ry 90 rz 0 deg; joints [-9.498, 5.066, 49.946, 168.458, 55.56, -173.412]
  Set speed (30.0 mm/s)
  Call Extruder(362.628)
  MoveL 601 to (44.51, 58.45, 1) mm, rotated rx 0 ry 90 rz 0 deg; joints [-10.525, 4.098, 52.615, 167.469, 57.343, -173.161]
  Set speed (90.0 mm/s)
  MoveL 602 to (45.64, 58.45, 1) mm, rotated rx 0 ry 90 rz 0 deg; joints [-10.512, 4.19, 52.359, 167.462, 57.181, -173.127]
  Set speed (30.0 mm/s)
  Call Extruder(365.038)
  MoveL 603 to (58.45, 45.64, 1) mm, rotated rx 0 ry 90 rz 0 deg; joints [-9.568, 5.083, 49.901, 168.37, 55.54, -173.357]
  Set speed (90.0 mm/s)
  MoveL 604 to (58.45, 46.77, 1) mm, rotated rx 0 ry 90 rz 0 deg; joints [-9.639, 5.1, 49.855, 168.281, 55.52, -173.302]
  Set speed (30.0 mm/s)
  Call Extruder(367.236)
  MoveL 605 to (46.77, 58.45, 1) mm, rotated rx 0 ry 90 rz 0 deg; joints [-10.499, 4.282, 52.101, 167.454, 57.019, -173.093]
  Set speed (90.0 mm/s)
  MoveL 606 to (47.9, 58.45, 1) mm, rotated rx 0 ry 90 rz 0 deg; joints [-10.485, 4.376, 51.842, 167.447, 56.856, -173.059]
  Set speed (30.0 mm/s)
  Call Extruder(369.221)
  MoveL 607 to (58.45, 47.9, 1) mm, rotated rx 0 ry 90 rz 0 deg; joints [-9.709, 5.117, 49.809, 168.192, 55.5, -173.247]
  Set speed (90.0 mm/s)
  MoveL 608 to (58.45, 49.03, 1) mm, rotated rx 0 ry 90 rz 0 deg; joints [-9.78, 5.134, 49.762, 168.103, 55.479, -173.191]
  Set speed (30.0 mm/s)
  Call Extruder(370.993)
  MoveL 609 to (49.03, 58.45, 1) mm, rotated rx 0 ry 90 rz 0 deg; joints [-10.472, 4.47, 51.582, 167.438, 56.692, -173.024]
  Set speed (90.0 mm/s)
  MoveL 610 to (50.16, 58.45, 1) mm, rotated rx 0 ry 90 rz 0 deg; joints [-10.459, 4.565, 51.321, 167.43, 56.528, -172.989]
  Set speed (30.0 mm/s)
  Call Extruder(372.553)
  MoveL 611 to (58.45, 50.16, 1) mm, rotated rx 0 ry 90 rz 0 deg; joints [-9.85, 5.151, 49.715, 168.014, 55.459, -173.136]
  Set speed (90.0 mm/s)
  MoveL 612 to (58.45, 51.29, 1) mm, rotated rx 0 ry 90 rz 0 deg; joints [-9.92, 5.169, 49.668, 167.925, 55.438, -173.08]
  Set speed (30.0 mm/s)
  Call Extruder(373.899)
  MoveL 613 to (51.29, 58.45, 1) mm, rotated rx 0 ry 90 rz 0 deg; joints [-10.446, 4.66, 51.058, 167.421, 56.363, -172.954]
  Set speed (90.0 mm/s)
  MoveL 614 to (52.42, 58.45, 1) mm, rotated rx 0 ry 90 rz 0 deg; joints [-10.433, 4.756, 50.793, 167.413, 56.197, -172.918]
  Set speed (30.0 mm/s)
  Call Extruder(375.032)
  MoveL 615 to (58.45, 52.42, 1) mm, rotated rx 0 ry 90 rz 0 deg; joints [-9.991, 5.186, 49.62, 167.835, 55.417, -173.024]
  Set speed (90.0 mm/s)
  MoveL 616 to (58.45, 53.56, 1) mm, rotated rx 0 ry 90 rz 0 deg; joints [-10.061, 5.204, 49.572, 167.746, 55.396, -172.968]
  Set speed (30.0 mm/s)
  Call Extruder(375.953)
  MoveL 617 to (53.56, 58.45, 1) mm, rotated rx 0 ry 90 rz 0 deg; joints [-10.42, 4.853, 50.527, 167.403, 56.03, -172.883]
  Set speed (90.0 mm/s)
  MoveL 618 to (54.69, 58.45, 1) mm, rotated rx 0 ry 90 rz 0 deg; joints [-10.407, 4.951, 50.26, 167.394, 55.863, -172.847]
  Set speed (30.0 mm/s)
  Call Extruder(376.661)
  MoveL 619 to (58.45, 54.69, 1) mm, rotated rx 0 ry 90 rz 0 deg; joints [-10.131, 5.222, 49.523, 167.657, 55.374, -172.912]
  Set speed (90.0 mm/s)
  MoveL 620 to (58.45, 55.82, 1) mm, rotated rx 0 ry 90 rz 0 deg; joints [-10.201, 5.24, 49.474, 167.568, 55.353, -172.856]
  Set speed (30.0 mm/s)
  Call Extruder(377.156)
  MoveL 621 to (55.82, 58.45, 1) mm, rotated rx 0 ry 90 rz 0 deg; joints [-10.394, 5.05, 49.99, 167.384, 55.695, -172.81]
  Set speed (90.0 mm/s)
  MoveL 622 to (56.95, 58.45, 1) mm, rotated rx 0 ry 90 rz 0 deg; joints [-10.382, 5.15, 49.72, 167.374, 55.527, -172.774]
  Set speed (30.0 mm/s)
  Call Extruder(377.438)
  MoveL 623 to (58.45, 56.95, 1) mm, rotated rx 0 ry 90 rz 0 deg; joints [-10.272, 5.258, 49.425, 167.478, 55.331, -172.8]
  Set speed (90.0 mm/s)
  MoveL 624 to (58.45, 58.08, 1) mm, rotated rx 0 ry 90 rz 0 deg; joints [-10.342, 5.277, 49.375, 167.389, 55.309, -172.743]
  Set speed (30.0 mm/s)
  Call Extruder(377.507)
  MoveL 625 to (58.08, 58.45, 1) mm, rotated rx 0 ry 90 rz 0 deg; joints [-10.369, 5.25, 49.448, 167.364, 55.357, -172.737]
  Set speed (90.0 mm/s)
  MoveL 626 to (52.43, 41.12, 1) mm, rotated rx 0 ry 90 rz 0 deg; joints [-9.348, 4.501, 51.496, 168.768, 56.508, -173.747]
  Set speed (120.0 mm/s)
  MoveL 627 to (52.43, 41.12, 1.4) mm, rotated rx 0 ry 90 rz 0 deg; joints [-9.348, 4.457, 51.544, 168.769, 56.513, -173.748]
  Set speed (60.0 mm/s)
  Call Extruder(378.720)
  MoveL 628 to (58.88, 47.57, 1.4) mm, rotated rx 0 ry 90 rz 0 deg; joints [-9.684, 5.106, 49.769, 168.215, 55.447, -173.251]
  Call Extruder(379.577)
  MoveL 629 to (58.88, 41.12, 1.4) mm, rotated rx 0 ry 90 rz 0 deg; joints [-9.282, 5.011, 50.027, 168.722, 55.561, -173.565]
  Call Extruder(382.919)
  MoveL 630 to (41.12, 58.88, 1.4) mm, rotated rx 0 ry 90 rz 0 deg; joints [-10.592, 3.79, 53.402, 167.457, 57.82, -173.242]
  Call Extruder(382.919)
  MoveL 631 to (41.12, 58.88, 1.4) mm, rotated rx 0 ry 90 rz 0 deg; joints [-10.592, 3.791, 53.402, 167.457, 57.82, -173.242]
  Call Extruder(383.777)
  MoveL 632 to (41.12, 52.43, 1.4) mm, rotated rx 0 ry 90 rz 0 deg; joints [-10.184, 3.697, 53.664, 167.957, 57.938, -173.539]
  Call Extruder(384.990)
  MoveL 633 to (47.57, 58.88, 1.4) mm, rotated rx 0 ry 90 rz 0 deg; joints [-10.516, 4.311, 51.949, 167.416, 56.9, -173.05]
  Call Extruder(385.637)
  MoveL 634 to (52.43, 58.88, 1.4) mm, rotated rx 0 ry 90 rz 0 deg; joints [-10.46, 4.72, 50.822, 167.379, 56.192, -172.899]
  Call Extruder(386.850)
  MoveL 635 to (58.88, 52.43, 1.4) mm, rotated rx 0 ry 90 rz 0 deg; joints [-9.986, 5.18, 49.566, 167.832, 55.357, -173.012]
  Call Extruder(387.708)
  MoveL 636 to (58.88, 58.88, 1.4) mm, rotated rx 0 ry 90 rz 0 deg; joints [-10.386, 5.284, 49.286, 167.323, 55.235, -172.691]
  Call Extruder(387.708)
  MoveL 637 to (58.88, 58.88, 1.4) mm, rotated rx 0 ry 90 rz 0 deg; joints [-10.386, 5.284, 49.286, 167.323, 55.235, -172.691]
  Call Extruder(391.049)
  MoveL 638 to (41.12, 41.12, 1.4) mm, rotated rx 0 ry 90 rz 0 deg; joints [-9.467, 3.544, 54.096, 168.833, 58.134, -174.05]
  Call Extruder(391.907)
  MoveL 639 to (41.12, 47.56, 1.4) mm, rotated rx 0 ry 90 rz 0 deg; joints [-9.876, 3.63, 53.854, 168.335, 58.024, -173.76]
  Call Extruder(393.120)
  MoveL 640 to (47.57, 41.12, 1.4) mm, rotated rx 0 ry 90 rz 0 deg; joints [-9.399, 4.056, 52.659, 168.799, 57.218, -173.88]
  Call Extruder(394.625)
